// TIA Portal V20 export
TYPE "type_emRelations_em5_cmStatus"
// stored: Access Published, Namespace Unit1
   STRUCT
      cmPnp1stCathodeDetect { S7_SetPoint := 'True'} : "LBC_typeDigitalSignalControlNode";
      cmPnp2ndCathodeDetect { S7_SetPoint := 'True'} : "LBC_typeDigitalSignalControlNode";
      cmCathodeAlignTableElectrodeDetect { S7_SetPoint := 'True'} : "LBC_typeDigitalSignalControlNode";
      cmCathodeNgPnpElectrodeDetect { S7_SetPoint := 'True'} : "LBC_typeDigitalSignalControlNode";
      cmCathodeNgBoxFullSensorDetect { S7_SetPoint := 'True'} : "LBC_typeDigitalSignalControlNode";
      cmCathodeNgBoxDetect { S7_SetPoint := 'True'} : "LBC_typeDigitalSignalControlNode";
      cmCathodeMainPnP1AxisX { ExternalAccessible := 'False'; ExternalVisible := 'False'; ExternalWritable := 'False'} : "LBC_typeAxis64PosControlNode";
      cmCathodeMainPnP2AxisX { ExternalAccessible := 'False'; ExternalVisible := 'False'; ExternalWritable := 'False'} : "LBC_typeAxis64PosControlNode";
      cmCathodeMainPnP1AxisY { ExternalAccessible := 'False'; ExternalVisible := 'False'; ExternalWritable := 'False'} : "LBC_typeAxis64PosControlNode";
      cmCathodeMainPnP1AxisZ { ExternalAccessible := 'False'; ExternalVisible := 'False'; ExternalWritable := 'False'} : "LBC_typeAxis64PosControlNode";
      cmCathodeMainPnP2AxisZ { ExternalAccessible := 'False'; ExternalVisible := 'False'; ExternalWritable := 'False'} : "LBC_typeAxis64PosControlNode";
      cmCathodeAlignTableAxisX { ExternalAccessible := 'False'; ExternalVisible := 'False'; ExternalWritable := 'False'} : "LBC_typeAxis64PosControlNode";
      cmCathodeAlignTableAxisY1 { ExternalAccessible := 'False'; ExternalVisible := 'False'; ExternalWritable := 'False'} : "LBC_typeAxis64PosControlNode";
      cmCathodeAlignTableAxisY2 { ExternalAccessible := 'False'; ExternalVisible := 'False'; ExternalWritable := 'False'} : "LBC_typeAxis64PosControlNode";
      cmCathodeMainPnP1RotaryCwCcw { ExternalAccessible := 'False'; ExternalVisible := 'False'; ExternalWritable := 'False'} : "LBC_typeTwoWayActuatorControlNode";
      cmCathodeMainPnP1SuctionPlateVacuum { ExternalAccessible := 'False'; ExternalVisible := 'False'; ExternalWritable := 'False'} : "LBC_typeTwoWayActuatorControlNode";
      cmCathodeMainPnP2SuctionPlateVacuum { ExternalAccessible := 'False'; ExternalVisible := 'False'; ExternalWritable := 'False'} : "LBC_typeTwoWayActuatorControlNode";
      cmCathodeAlignTableSuctionPlateVacuum { ExternalAccessible := 'False'; ExternalVisible := 'False'; ExternalWritable := 'False'} : "LBC_typeTwoWayActuatorControlNode";
      cmCathodeGlassCleaning { ExternalAccessible := 'False'; ExternalVisible := 'False'; ExternalWritable := 'False'} : "LBC_typeTwoWayActuatorControlNode";
      cmCathodeNgPnpUpDown { ExternalAccessible := 'False'; ExternalVisible := 'False'; ExternalWritable := 'False'} : "LBC_typeTwoWayActuatorControlNode";
      cmCathodeNgPnp1stFwdBwd { ExternalAccessible := 'False'; ExternalVisible := 'False'; ExternalWritable := 'False'} : "LBC_typeTwoWayActuatorControlNode";
      cmCathodeNgPnp2ndFwdBwd { ExternalAccessible := 'False'; ExternalVisible := 'False'; ExternalWritable := 'False'; S7_SetPoint := 'True'} : "LBC_typeTwoWayActuatorControlNode";
      cmCathodeMaintenanceMovingFixFwdBwd { ExternalAccessible := 'False'; ExternalVisible := 'False'; ExternalWritable := 'False'} : "LBC_typeTwoWayActuatorControlNode";
      cmCathodeNgBoxLiftUpDown { ExternalAccessible := 'False'; ExternalVisible := 'False'; ExternalWritable := 'False'; S7_SetPoint := 'True'} : "LBC_typeTwoWayActuatorControlNode";
      cmCathodeNgBoxLockUpDown { ExternalAccessible := 'False'; ExternalVisible := 'False'; ExternalWritable := 'False'; S7_SetPoint := 'True'} : "LBC_typeTwoWayActuatorControlNode";
      cmCathodeNgPnpVaccum { ExternalAccessible := 'False'; ExternalVisible := 'False'; ExternalWritable := 'False'} : "LBC_typeTwoWayActuatorControlNode";
      cmCathodeConveyorCoverFwdBwd { S7_SetPoint := 'True'} : "LBC_typeTwoWayActuatorControlNode";
      cmCathodeConveyorPickUpBlower { S7_SetPoint := 'True'} : "LBC_typeTwoWayActuatorControlNode";
      cmCathodeVisionControllerInterface { ExternalAccessible := 'False'; ExternalVisible := 'False'; ExternalWritable := 'False'} : "LER_typeVisionControlNode";
   END_STRUCT;
   // cmPnp1stCathodeDetect.commands.reset := FALSE;
   // cmPnp1stCathodeDetect.commands.simulation := FALSE;
   // cmPnp1stCathodeDetect.commands.quality := TRUE;
   // cmPnp1stCathodeDetect.monitoring.valid := TRUE;
   // cmPnp1stCathodeDetect.monitoring.busy := TRUE;
   // cmPnp1stCathodeDetect.monitoring.error := FALSE;
   // cmPnp1stCathodeDetect.monitoring.status := 16#0000;
   // cmPnp1stCathodeDetect.monitoring.risingEdge := FALSE;
   // cmPnp1stCathodeDetect.monitoring.fallingEdge := FALSE;
   // cmPnp1stCathodeDetect.monitoring.processValue := FALSE;
   // cmPnp2ndCathodeDetect.commands.reset := FALSE;
   // cmPnp2ndCathodeDetect.commands.simulation := FALSE;
   // cmPnp2ndCathodeDetect.commands.quality := TRUE;
   // cmPnp2ndCathodeDetect.monitoring.valid := TRUE;
   // cmPnp2ndCathodeDetect.monitoring.busy := TRUE;
   // cmPnp2ndCathodeDetect.monitoring.error := FALSE;
   // cmPnp2ndCathodeDetect.monitoring.status := 16#0000;
   // cmPnp2ndCathodeDetect.monitoring.risingEdge := FALSE;
   // cmPnp2ndCathodeDetect.monitoring.fallingEdge := FALSE;
   // cmPnp2ndCathodeDetect.monitoring.processValue := FALSE;
   // cmCathodeAlignTableElectrodeDetect.commands.reset := FALSE;
   // cmCathodeAlignTableElectrodeDetect.commands.simulation := FALSE;
   // cmCathodeAlignTableElectrodeDetect.commands.quality := TRUE;
   // cmCathodeAlignTableElectrodeDetect.monitoring.valid := TRUE;
   // cmCathodeAlignTableElectrodeDetect.monitoring.busy := TRUE;
   // cmCathodeAlignTableElectrodeDetect.monitoring.error := FALSE;
   // cmCathodeAlignTableElectrodeDetect.monitoring.status := 16#0000;
   // cmCathodeAlignTableElectrodeDetect.monitoring.risingEdge := FALSE;
   // cmCathodeAlignTableElectrodeDetect.monitoring.fallingEdge := FALSE;
   // cmCathodeAlignTableElectrodeDetect.monitoring.processValue := FALSE;
   // cmCathodeNgPnpElectrodeDetect.commands.reset := FALSE;
   // cmCathodeNgPnpElectrodeDetect.commands.simulation := FALSE;
   // cmCathodeNgPnpElectrodeDetect.commands.quality := TRUE;
   // cmCathodeNgPnpElectrodeDetect.monitoring.valid := FALSE;
   // cmCathodeNgPnpElectrodeDetect.monitoring.busy := FALSE;
   // cmCathodeNgPnpElectrodeDetect.monitoring.error := FALSE;
   // cmCathodeNgPnpElectrodeDetect.monitoring.status := 16#0000;
   // cmCathodeNgPnpElectrodeDetect.monitoring.risingEdge := FALSE;
   // cmCathodeNgPnpElectrodeDetect.monitoring.fallingEdge := FALSE;
   // cmCathodeNgPnpElectrodeDetect.monitoring.processValue := FALSE;
   // cmCathodeNgBoxFullSensorDetect.commands.reset := FALSE;
   // cmCathodeNgBoxFullSensorDetect.commands.simulation := FALSE;
   // cmCathodeNgBoxFullSensorDetect.commands.quality := TRUE;
   // cmCathodeNgBoxFullSensorDetect.monitoring.valid := TRUE;
   // cmCathodeNgBoxFullSensorDetect.monitoring.busy := TRUE;
   // cmCathodeNgBoxFullSensorDetect.monitoring.error := FALSE;
   // cmCathodeNgBoxFullSensorDetect.monitoring.status := 16#0000;
   // cmCathodeNgBoxFullSensorDetect.monitoring.risingEdge := FALSE;
   // cmCathodeNgBoxFullSensorDetect.monitoring.fallingEdge := FALSE;
   // cmCathodeNgBoxFullSensorDetect.monitoring.processValue := FALSE;
   // cmCathodeNgBoxDetect.commands.reset := FALSE;
   // cmCathodeNgBoxDetect.commands.simulation := FALSE;
   // cmCathodeNgBoxDetect.commands.quality := TRUE;
   // cmCathodeNgBoxDetect.monitoring.valid := TRUE;
   // cmCathodeNgBoxDetect.monitoring.busy := TRUE;
   // cmCathodeNgBoxDetect.monitoring.error := FALSE;
   // cmCathodeNgBoxDetect.monitoring.status := 16#0000;
   // cmCathodeNgBoxDetect.monitoring.risingEdge := FALSE;
   // cmCathodeNgBoxDetect.monitoring.fallingEdge := FALSE;
   // cmCathodeNgBoxDetect.monitoring.processValue := TRUE;
   // cmCathodeMainPnP1AxisX.commandConfiguration.generalSettings.stopOnError := TRUE;
   // cmCathodeMainPnP1AxisX.commandConfiguration.generalSettings.resetWithRestart := FALSE;
   // cmCathodeMainPnP1AxisX.commandConfiguration.generalSettings.abortWaitingSyncCmd := TRUE;
   // cmCathodeMainPnP1AxisX.commandConfiguration.power.startMode := 1;
   // cmCathodeMainPnP1AxisX.commandConfiguration.power.stopMode := 0;
   // cmCathodeMainPnP1AxisX.commandConfiguration.power.syncMotionSimulation := FALSE;
   // cmCathodeMainPnP1AxisX.commandConfiguration.power.syncMotionSimulationExtendedMode := -1;
   // cmCathodeMainPnP1AxisX.commandConfiguration.jog.velocity := 0.0;
   // cmCathodeMainPnP1AxisX.commandConfiguration.jog.acceleration := -1.0;
   // cmCathodeMainPnP1AxisX.commandConfiguration.jog.deceleration := -1.0;
   // cmCathodeMainPnP1AxisX.commandConfiguration.jog.jerk := -1.0;
   // cmCathodeMainPnP1AxisX.commandConfiguration.jog.positionControlled := TRUE;
   // cmCathodeMainPnP1AxisX.commandConfiguration.jog.increment := 0.0;
   // cmCathodeMainPnP1AxisX.commandConfiguration.jog.mode := 0;
   // cmCathodeMainPnP1AxisX.commandConfiguration.moveVelocity.velocity := 0.0;
   // cmCathodeMainPnP1AxisX.commandConfiguration.moveVelocity.acceleration := -1.0;
   // cmCathodeMainPnP1AxisX.commandConfiguration.moveVelocity.deceleration := -1.0;
   // cmCathodeMainPnP1AxisX.commandConfiguration.moveVelocity.jerk := -1.0;
   // cmCathodeMainPnP1AxisX.commandConfiguration.moveVelocity.direction := 0;
   // cmCathodeMainPnP1AxisX.commandConfiguration.moveVelocity.positionControlled := TRUE;
   // cmCathodeMainPnP1AxisX.commandConfiguration.moveVelocity.velocityChangeOnTheFly := FALSE;
   // cmCathodeMainPnP1AxisX.commandConfiguration.stop.deceleration := -1.0;
   // cmCathodeMainPnP1AxisX.commandConfiguration.stop.jerk := -1.0;
   // cmCathodeMainPnP1AxisX.commandConfiguration.stop.abortAcceleration := FALSE;
   // cmCathodeMainPnP1AxisX.commandConfiguration.fastStop.deceleration := -1.0;
   // cmCathodeMainPnP1AxisX.commandConfiguration.fastStop.jerk := -1.0;
   // cmCathodeMainPnP1AxisX.commandConfiguration.fastStop.abortAcceleration := FALSE;
   // cmCathodeMainPnP1AxisX.commandConfiguration.fastStop.replaceStopPossible := FALSE;
   // cmCathodeMainPnP1AxisX.commandConfiguration.torqueLimiting.limit := -1.0;
   // cmCathodeMainPnP1AxisX.commandConfiguration.torqueLimiting.mode := 0;
   // cmCathodeMainPnP1AxisX.commandConfiguration.homing.position := 0.0;
   // cmCathodeMainPnP1AxisX.commandConfiguration.homing.mode := 0;
   // cmCathodeMainPnP1AxisX.commandConfiguration.homing.sensor := 0;
   // cmCathodeMainPnP1AxisX.commandConfiguration.homing.extendedMode := -1;
   // cmCathodeMainPnP1AxisX.commandConfiguration.homing.extendedModeTorqueLimit := 0.0;
   // cmCathodeMainPnP1AxisX.commandConfiguration.homing.extendedModeTargetPosition := 0.0;
   // cmCathodeMainPnP1AxisX.commandConfiguration.posRelative.distance := 0.0;
   // cmCathodeMainPnP1AxisX.commandConfiguration.posRelative.velocity := -1.0;
   // cmCathodeMainPnP1AxisX.commandConfiguration.posRelative.acceleration := -1.0;
   // cmCathodeMainPnP1AxisX.commandConfiguration.posRelative.deceleration := -1.0;
   // cmCathodeMainPnP1AxisX.commandConfiguration.posRelative.jerk := -1.0;
   // cmCathodeMainPnP1AxisX.commandConfiguration.posRelative.direction := 0;
   // cmCathodeMainPnP1AxisX.commandConfiguration.posAbsolute.position := 0.0;
   // cmCathodeMainPnP1AxisX.commandConfiguration.posAbsolute.velocity := -1.0;
   // cmCathodeMainPnP1AxisX.commandConfiguration.posAbsolute.acceleration := -1.0;
   // cmCathodeMainPnP1AxisX.commandConfiguration.posAbsolute.deceleration := -1.0;
   // cmCathodeMainPnP1AxisX.commandConfiguration.posAbsolute.jerk := -1.0;
   // cmCathodeMainPnP1AxisX.commandConfiguration.posAbsolute.direction := 1;
   // cmCathodeMainPnP1AxisX.commandConfiguration.posAbsolute.positionChangeOnTheFly := FALSE;
   // cmCathodeMainPnP1AxisX.commandConfiguration.posAbsolute.velocityChangeOnTheFly := FALSE;
   // cmCathodeMainPnP1AxisX.commandConfiguration.posSuperimposed.distance := 0.0;
   // cmCathodeMainPnP1AxisX.commandConfiguration.posSuperimposed.velocityDiff := -1.0;
   // cmCathodeMainPnP1AxisX.commandConfiguration.posSuperimposed.acceleration := -1.0;
   // cmCathodeMainPnP1AxisX.commandConfiguration.posSuperimposed.deceleration := -1.0;
   // cmCathodeMainPnP1AxisX.commandConfiguration.posSuperimposed.jerk := -1.0;
   // cmCathodeMainPnP1AxisX.commandConfiguration.posSuperimposed.direction := 0;
   // cmCathodeMainPnP1AxisX.commandConfiguration.haltSuperimposed.deceleration := -1.0;
   // cmCathodeMainPnP1AxisX.commandConfiguration.haltSuperimposed.jerk := -1.0;
   // cmCathodeMainPnP1AxisX.commandConfiguration.haltSuperimposed.abortAcceleration := FALSE;
   // cmCathodeMainPnP1AxisX.commandConfiguration.gearInRelative.ratioNumerator := 1;
   // cmCathodeMainPnP1AxisX.commandConfiguration.gearInRelative.ratioDenominator := 1;
   // cmCathodeMainPnP1AxisX.commandConfiguration.gearInRelative.acceleration := -1.0;
   // cmCathodeMainPnP1AxisX.commandConfiguration.gearInRelative.deceleration := -1.0;
   // cmCathodeMainPnP1AxisX.commandConfiguration.gearInRelative.jerk := -1.0;
   // cmCathodeMainPnP1AxisX.commandConfiguration.gearInRelative.ratioChangeOnTheFly := FALSE;
   // cmCathodeMainPnP1AxisX.commandConfiguration.gearInAbsolute.ratioNumerator := 1;
   // cmCathodeMainPnP1AxisX.commandConfiguration.gearInAbsolute.ratioDenominator := 1;
   // cmCathodeMainPnP1AxisX.commandConfiguration.gearInAbsolute.masterSyncPosition := 0.0;
   // cmCathodeMainPnP1AxisX.commandConfiguration.gearInAbsolute.slaveSyncPosition := 0.0;
   // cmCathodeMainPnP1AxisX.commandConfiguration.gearInAbsolute.syncProfileReference := 1;
   // cmCathodeMainPnP1AxisX.commandConfiguration.gearInAbsolute.masterStartDistance := 0.0;
   // cmCathodeMainPnP1AxisX.commandConfiguration.gearInAbsolute.velocity := -1.0;
   // cmCathodeMainPnP1AxisX.commandConfiguration.gearInAbsolute.acceleration := -1.0;
   // cmCathodeMainPnP1AxisX.commandConfiguration.gearInAbsolute.deceleration := -1.0;
   // cmCathodeMainPnP1AxisX.commandConfiguration.gearInAbsolute.jerk := -1.0;
   // cmCathodeMainPnP1AxisX.commandConfiguration.gearInAbsolute.syncDirection := 1;
   // cmCathodeMainPnP1AxisX.commandConfiguration.gearInAbsolute.ratioChangeOnTheFly := FALSE;
   // cmCathodeMainPnP1AxisX.commandConfiguration.gearInVelocity.continuousUpdate := FALSE;
   // cmCathodeMainPnP1AxisX.commandConfiguration.gearInVelocity.ratioNumerator := 1;
   // cmCathodeMainPnP1AxisX.commandConfiguration.gearInVelocity.ratioDenominator := 1;
   // cmCathodeMainPnP1AxisX.commandConfiguration.gearInVelocity.acceleration := -1.0;
   // cmCathodeMainPnP1AxisX.commandConfiguration.gearInVelocity.deceleration := -1.0;
   // cmCathodeMainPnP1AxisX.commandConfiguration.gearInVelocity.jerk := -1.0;
   // cmCathodeMainPnP1AxisX.commandConfiguration.gearInVelocity.positionControlled := FALSE;
   // cmCathodeMainPnP1AxisX.commandConfiguration.camIn.masterOffset := 0.0;
   // cmCathodeMainPnP1AxisX.commandConfiguration.camIn.slaveOffset := 0.0;
   // cmCathodeMainPnP1AxisX.commandConfiguration.camIn.masterScaling := 1.0;
   // cmCathodeMainPnP1AxisX.commandConfiguration.camIn.slaveScaling := 1.0;
   // cmCathodeMainPnP1AxisX.commandConfiguration.camIn.masterSyncPosition := 0.0;
   // cmCathodeMainPnP1AxisX.commandConfiguration.camIn.syncProfileReference := 1;
   // cmCathodeMainPnP1AxisX.commandConfiguration.camIn.masterStartDistance := 0.0;
   // cmCathodeMainPnP1AxisX.commandConfiguration.camIn.velocity := -1.0;
   // cmCathodeMainPnP1AxisX.commandConfiguration.camIn.acceleration := -1.0;
   // cmCathodeMainPnP1AxisX.commandConfiguration.camIn.deceleration := -1.0;
   // cmCathodeMainPnP1AxisX.commandConfiguration.camIn.jerk := -1.0;
   // cmCathodeMainPnP1AxisX.commandConfiguration.camIn.applicationMode := 0;
   // cmCathodeMainPnP1AxisX.commandConfiguration.camIn.syncDirection := 1;
   // cmCathodeMainPnP1AxisX.commandConfiguration.gearOutCamOut.slavePosition := 0.0;
   // cmCathodeMainPnP1AxisX.commandConfiguration.gearOutCamOut.syncProfileReference := 1;
   // cmCathodeMainPnP1AxisX.commandConfiguration.gearOutCamOut.masterStopDistance := 0.0;
   // cmCathodeMainPnP1AxisX.commandConfiguration.gearOutCamOut.deceleration := -1.0;
   // cmCathodeMainPnP1AxisX.commandConfiguration.gearOutCamOut.jerk := -1.0;
   // cmCathodeMainPnP1AxisX.commandConfiguration.gearOutCamOut.syncOutDirection := 3;
   // cmCathodeMainPnP1AxisX.commandConfiguration.gearOutCamOut.gearOutCamOutMode := -1;
   // cmCathodeMainPnP1AxisX.commandConfiguration.phasing.phaseShift := 0.0;
   // cmCathodeMainPnP1AxisX.commandConfiguration.phasing.velocity := -1.0;
   // cmCathodeMainPnP1AxisX.commandConfiguration.phasing.acceleration := -1.0;
   // cmCathodeMainPnP1AxisX.commandConfiguration.phasing.deceleration := -1.0;
   // cmCathodeMainPnP1AxisX.commandConfiguration.phasing.jerk := -1.0;
   // cmCathodeMainPnP1AxisX.commandConfiguration.phasing.profileReference := 0;
   // cmCathodeMainPnP1AxisX.commandConfiguration.phasing.phasingDistance := 0.0;
   // cmCathodeMainPnP1AxisX.commandConfiguration.phasing.startPosition := 0.0;
   // cmCathodeMainPnP1AxisX.commandConfiguration.phasing.direction := 3;
   // cmCathodeMainPnP1AxisX.commandConfiguration.phasing.phaseAbsolute := TRUE;
   // cmCathodeMainPnP1AxisX.commandConfiguration.phasing.phaseShiftChangeOnTheFly := FALSE;
   // cmCathodeMainPnP1AxisX.commandConfiguration.offset.offset := 0.0;
   // cmCathodeMainPnP1AxisX.commandConfiguration.offset.profileReference := 1;
   // cmCathodeMainPnP1AxisX.commandConfiguration.offset.offsetDistance := 0.0;
   // cmCathodeMainPnP1AxisX.commandConfiguration.offset.startPosition := 0.0;
   // cmCathodeMainPnP1AxisX.commandConfiguration.offset.direction := 3;
   // cmCathodeMainPnP1AxisX.commandConfiguration.offset.offsetAbsolute := TRUE;
   // cmCathodeMainPnP1AxisX.commandConfiguration.offset.offsetChangeOnTheFly := FALSE;
   // cmCathodeMainPnP1AxisX.commands.enableAxis := FALSE;
   // cmCathodeMainPnP1AxisX.commands.resetAxis := FALSE;
   // cmCathodeMainPnP1AxisX.commands.openBrake := FALSE;
   // cmCathodeMainPnP1AxisX.commands.jogForward := FALSE;
   // cmCathodeMainPnP1AxisX.commands.jogBackward := FALSE;
   // cmCathodeMainPnP1AxisX.commands.moveVelocity := FALSE;
   // cmCathodeMainPnP1AxisX.commands.stop := FALSE;
   // cmCathodeMainPnP1AxisX.commands.fastStop := FALSE;
   // cmCathodeMainPnP1AxisX.commands.torqueLimiting := FALSE;
   // cmCathodeMainPnP1AxisX.commands.homing := FALSE;
   // cmCathodeMainPnP1AxisX.commands.posRelative := FALSE;
   // cmCathodeMainPnP1AxisX.commands.posAbsolute := FALSE;
   // cmCathodeMainPnP1AxisX.commands.posSuperimposed := FALSE;
   // cmCathodeMainPnP1AxisX.commands.haltSuperimposed := FALSE;
   // cmCathodeMainPnP1AxisX.commands.selectSetPosition := -1;
   // cmCathodeMainPnP1AxisX.commands.reset := FALSE;
   // cmCathodeMainPnP1AxisX.monitoring.valid := FALSE;
   // cmCathodeMainPnP1AxisX.monitoring.busy := TRUE;
   // cmCathodeMainPnP1AxisX.monitoring.error := TRUE;
   // cmCathodeMainPnP1AxisX.monitoring.status := 16#8600;
   // cmCathodeMainPnP1AxisX.monitoring.subfunctionStatus := 16#8001;
   // cmCathodeMainPnP1AxisX.monitoring.axisEnabled := FALSE;
   // cmCathodeMainPnP1AxisX.monitoring.resetActive := FALSE;
   // cmCathodeMainPnP1AxisX.monitoring.inVelocity := FALSE;
   // cmCathodeMainPnP1AxisX.monitoring.inLimitation := FALSE;
   // cmCathodeMainPnP1AxisX.monitoring.inClamping := FALSE;
   // cmCathodeMainPnP1AxisX.monitoring.startSync := FALSE;
   // cmCathodeMainPnP1AxisX.monitoring.inSync := FALSE;
   // cmCathodeMainPnP1AxisX.monitoring.inSimulation := FALSE;
   // cmCathodeMainPnP1AxisX.monitoring.jogSelected := FALSE;
   // cmCathodeMainPnP1AxisX.monitoring.moveVelocitySelected := FALSE;
   // cmCathodeMainPnP1AxisX.monitoring.stopSelected := FALSE;
   // cmCathodeMainPnP1AxisX.monitoring.fastStopSelected := FALSE;
   // cmCathodeMainPnP1AxisX.monitoring.torqueLimitingSelected := FALSE;
   // cmCathodeMainPnP1AxisX.monitoring.homingSelected := FALSE;
   // cmCathodeMainPnP1AxisX.monitoring.posRelativeSelected := FALSE;
   // cmCathodeMainPnP1AxisX.monitoring.posAbsoluteSelected := FALSE;
   // cmCathodeMainPnP1AxisX.monitoring.posSuperimposedSelected := FALSE;
   // cmCathodeMainPnP1AxisX.monitoring.haltSuperimposedSelected := FALSE;
   // cmCathodeMainPnP1AxisX.monitoring.commandBusy := FALSE;
   // cmCathodeMainPnP1AxisX.monitoring.commandDone := FALSE;
   // cmCathodeMainPnP1AxisX.monitoring.commandAborted := FALSE;
   // cmCathodeMainPnP1AxisX.monitoring.homingCommandBusy := FALSE;
   // cmCathodeMainPnP1AxisX.monitoring.homingCommandDone := FALSE;
   // cmCathodeMainPnP1AxisX.monitoring.homingCommandAborted := FALSE;
   // cmCathodeMainPnP1AxisX.monitoring.superimposedBusy := FALSE;
   // cmCathodeMainPnP1AxisX.monitoring.superimposedDone := FALSE;
   // cmCathodeMainPnP1AxisX.monitoring.superimposedAborted := FALSE;
   // cmCathodeMainPnP1AxisX.monitoring.actualPosition := 0.048;
   // cmCathodeMainPnP1AxisX.monitoring.actualSpeed := 0.0;
   // cmCathodeMainPnP1AxisX.monitoring.speedUnit := 1062;
   // cmCathodeMainPnP1AxisX.monitoring.positionUnit := 1013;
   // cmCathodeMainPnP1AxisX.monitoring.axisType := 1;
   // cmCathodeMainPnP1AxisX.monitoring.interlockGeneralOut := TRUE;
   // cmCathodeMainPnP1AxisX.monitoring.interlockJogForwardOut := TRUE;
   // cmCathodeMainPnP1AxisX.monitoring.interlockJogBackwardOut := TRUE;
   // cmCathodeMainPnP2AxisX.commandConfiguration.generalSettings.stopOnError := TRUE;
   // cmCathodeMainPnP2AxisX.commandConfiguration.generalSettings.resetWithRestart := FALSE;
   // cmCathodeMainPnP2AxisX.commandConfiguration.generalSettings.abortWaitingSyncCmd := TRUE;
   // cmCathodeMainPnP2AxisX.commandConfiguration.power.startMode := 1;
   // cmCathodeMainPnP2AxisX.commandConfiguration.power.stopMode := 0;
   // cmCathodeMainPnP2AxisX.commandConfiguration.power.syncMotionSimulation := FALSE;
   // cmCathodeMainPnP2AxisX.commandConfiguration.power.syncMotionSimulationExtendedMode := -1;
   // cmCathodeMainPnP2AxisX.commandConfiguration.jog.velocity := 0.0;
   // cmCathodeMainPnP2AxisX.commandConfiguration.jog.acceleration := -1.0;
   // cmCathodeMainPnP2AxisX.commandConfiguration.jog.deceleration := -1.0;
   // cmCathodeMainPnP2AxisX.commandConfiguration.jog.jerk := -1.0;
   // cmCathodeMainPnP2AxisX.commandConfiguration.jog.positionControlled := TRUE;
   // cmCathodeMainPnP2AxisX.commandConfiguration.jog.increment := 0.0;
   // cmCathodeMainPnP2AxisX.commandConfiguration.jog.mode := 0;
   // cmCathodeMainPnP2AxisX.commandConfiguration.moveVelocity.velocity := 0.0;
   // cmCathodeMainPnP2AxisX.commandConfiguration.moveVelocity.acceleration := -1.0;
   // cmCathodeMainPnP2AxisX.commandConfiguration.moveVelocity.deceleration := -1.0;
   // cmCathodeMainPnP2AxisX.commandConfiguration.moveVelocity.jerk := -1.0;
   // cmCathodeMainPnP2AxisX.commandConfiguration.moveVelocity.direction := 0;
   // cmCathodeMainPnP2AxisX.commandConfiguration.moveVelocity.positionControlled := TRUE;
   // cmCathodeMainPnP2AxisX.commandConfiguration.moveVelocity.velocityChangeOnTheFly := FALSE;
   // cmCathodeMainPnP2AxisX.commandConfiguration.stop.deceleration := -1.0;
   // cmCathodeMainPnP2AxisX.commandConfiguration.stop.jerk := -1.0;
   // cmCathodeMainPnP2AxisX.commandConfiguration.stop.abortAcceleration := FALSE;
   // cmCathodeMainPnP2AxisX.commandConfiguration.fastStop.deceleration := -1.0;
   // cmCathodeMainPnP2AxisX.commandConfiguration.fastStop.jerk := -1.0;
   // cmCathodeMainPnP2AxisX.commandConfiguration.fastStop.abortAcceleration := FALSE;
   // cmCathodeMainPnP2AxisX.commandConfiguration.fastStop.replaceStopPossible := FALSE;
   // cmCathodeMainPnP2AxisX.commandConfiguration.torqueLimiting.limit := -1.0;
   // cmCathodeMainPnP2AxisX.commandConfiguration.torqueLimiting.mode := 0;
   // cmCathodeMainPnP2AxisX.commandConfiguration.homing.position := 0.0;
   // cmCathodeMainPnP2AxisX.commandConfiguration.homing.mode := 0;
   // cmCathodeMainPnP2AxisX.commandConfiguration.homing.sensor := 0;
   // cmCathodeMainPnP2AxisX.commandConfiguration.homing.extendedMode := -1;
   // cmCathodeMainPnP2AxisX.commandConfiguration.homing.extendedModeTorqueLimit := 0.0;
   // cmCathodeMainPnP2AxisX.commandConfiguration.homing.extendedModeTargetPosition := 0.0;
   // cmCathodeMainPnP2AxisX.commandConfiguration.posRelative.distance := 0.0;
   // cmCathodeMainPnP2AxisX.commandConfiguration.posRelative.velocity := -1.0;
   // cmCathodeMainPnP2AxisX.commandConfiguration.posRelative.acceleration := -1.0;
   // cmCathodeMainPnP2AxisX.commandConfiguration.posRelative.deceleration := -1.0;
   // cmCathodeMainPnP2AxisX.commandConfiguration.posRelative.jerk := -1.0;
   // cmCathodeMainPnP2AxisX.commandConfiguration.posRelative.direction := 0;
   // cmCathodeMainPnP2AxisX.commandConfiguration.posAbsolute.position := 0.0;
   // cmCathodeMainPnP2AxisX.commandConfiguration.posAbsolute.velocity := -1.0;
   // cmCathodeMainPnP2AxisX.commandConfiguration.posAbsolute.acceleration := -1.0;
   // cmCathodeMainPnP2AxisX.commandConfiguration.posAbsolute.deceleration := -1.0;
   // cmCathodeMainPnP2AxisX.commandConfiguration.posAbsolute.jerk := -1.0;
   // cmCathodeMainPnP2AxisX.commandConfiguration.posAbsolute.direction := 1;
   // cmCathodeMainPnP2AxisX.commandConfiguration.posAbsolute.positionChangeOnTheFly := FALSE;
   // cmCathodeMainPnP2AxisX.commandConfiguration.posAbsolute.velocityChangeOnTheFly := FALSE;
   // cmCathodeMainPnP2AxisX.commandConfiguration.posSuperimposed.distance := 0.0;
   // cmCathodeMainPnP2AxisX.commandConfiguration.posSuperimposed.velocityDiff := -1.0;
   // cmCathodeMainPnP2AxisX.commandConfiguration.posSuperimposed.acceleration := -1.0;
   // cmCathodeMainPnP2AxisX.commandConfiguration.posSuperimposed.deceleration := -1.0;
   // cmCathodeMainPnP2AxisX.commandConfiguration.posSuperimposed.jerk := -1.0;
   // cmCathodeMainPnP2AxisX.commandConfiguration.posSuperimposed.direction := 0;
   // cmCathodeMainPnP2AxisX.commandConfiguration.haltSuperimposed.deceleration := -1.0;
   // cmCathodeMainPnP2AxisX.commandConfiguration.haltSuperimposed.jerk := -1.0;
   // cmCathodeMainPnP2AxisX.commandConfiguration.haltSuperimposed.abortAcceleration := FALSE;
   // cmCathodeMainPnP2AxisX.commandConfiguration.gearInRelative.ratioNumerator := 1;
   // cmCathodeMainPnP2AxisX.commandConfiguration.gearInRelative.ratioDenominator := 1;
   // cmCathodeMainPnP2AxisX.commandConfiguration.gearInRelative.acceleration := -1.0;
   // cmCathodeMainPnP2AxisX.commandConfiguration.gearInRelative.deceleration := -1.0;
   // cmCathodeMainPnP2AxisX.commandConfiguration.gearInRelative.jerk := -1.0;
   // cmCathodeMainPnP2AxisX.commandConfiguration.gearInRelative.ratioChangeOnTheFly := FALSE;
   // cmCathodeMainPnP2AxisX.commandConfiguration.gearInAbsolute.ratioNumerator := 1;
   // cmCathodeMainPnP2AxisX.commandConfiguration.gearInAbsolute.ratioDenominator := 1;
   // cmCathodeMainPnP2AxisX.commandConfiguration.gearInAbsolute.masterSyncPosition := 0.0;
   // cmCathodeMainPnP2AxisX.commandConfiguration.gearInAbsolute.slaveSyncPosition := 0.0;
   // cmCathodeMainPnP2AxisX.commandConfiguration.gearInAbsolute.syncProfileReference := 1;
   // cmCathodeMainPnP2AxisX.commandConfiguration.gearInAbsolute.masterStartDistance := 0.0;
   // cmCathodeMainPnP2AxisX.commandConfiguration.gearInAbsolute.velocity := -1.0;
   // cmCathodeMainPnP2AxisX.commandConfiguration.gearInAbsolute.acceleration := -1.0;
   // cmCathodeMainPnP2AxisX.commandConfiguration.gearInAbsolute.deceleration := -1.0;
   // cmCathodeMainPnP2AxisX.commandConfiguration.gearInAbsolute.jerk := -1.0;
   // cmCathodeMainPnP2AxisX.commandConfiguration.gearInAbsolute.syncDirection := 1;
   // cmCathodeMainPnP2AxisX.commandConfiguration.gearInAbsolute.ratioChangeOnTheFly := FALSE;
   // cmCathodeMainPnP2AxisX.commandConfiguration.gearInVelocity.continuousUpdate := FALSE;
   // cmCathodeMainPnP2AxisX.commandConfiguration.gearInVelocity.ratioNumerator := 1;
   // cmCathodeMainPnP2AxisX.commandConfiguration.gearInVelocity.ratioDenominator := 1;
   // cmCathodeMainPnP2AxisX.commandConfiguration.gearInVelocity.acceleration := -1.0;
   // cmCathodeMainPnP2AxisX.commandConfiguration.gearInVelocity.deceleration := -1.0;
   // cmCathodeMainPnP2AxisX.commandConfiguration.gearInVelocity.jerk := -1.0;
   // cmCathodeMainPnP2AxisX.commandConfiguration.gearInVelocity.positionControlled := FALSE;
   // cmCathodeMainPnP2AxisX.commandConfiguration.camIn.masterOffset := 0.0;
   // cmCathodeMainPnP2AxisX.commandConfiguration.camIn.slaveOffset := 0.0;
   // cmCathodeMainPnP2AxisX.commandConfiguration.camIn.masterScaling := 1.0;
   // cmCathodeMainPnP2AxisX.commandConfiguration.camIn.slaveScaling := 1.0;
   // cmCathodeMainPnP2AxisX.commandConfiguration.camIn.masterSyncPosition := 0.0;
   // cmCathodeMainPnP2AxisX.commandConfiguration.camIn.syncProfileReference := 1;
   // cmCathodeMainPnP2AxisX.commandConfiguration.camIn.masterStartDistance := 0.0;
   // cmCathodeMainPnP2AxisX.commandConfiguration.camIn.velocity := -1.0;
   // cmCathodeMainPnP2AxisX.commandConfiguration.camIn.acceleration := -1.0;
   // cmCathodeMainPnP2AxisX.commandConfiguration.camIn.deceleration := -1.0;
   // cmCathodeMainPnP2AxisX.commandConfiguration.camIn.jerk := -1.0;
   // cmCathodeMainPnP2AxisX.commandConfiguration.camIn.applicationMode := 0;
   // cmCathodeMainPnP2AxisX.commandConfiguration.camIn.syncDirection := 1;
   // cmCathodeMainPnP2AxisX.commandConfiguration.gearOutCamOut.slavePosition := 0.0;
   // cmCathodeMainPnP2AxisX.commandConfiguration.gearOutCamOut.syncProfileReference := 1;
   // cmCathodeMainPnP2AxisX.commandConfiguration.gearOutCamOut.masterStopDistance := 0.0;
   // cmCathodeMainPnP2AxisX.commandConfiguration.gearOutCamOut.deceleration := -1.0;
   // cmCathodeMainPnP2AxisX.commandConfiguration.gearOutCamOut.jerk := -1.0;
   // cmCathodeMainPnP2AxisX.commandConfiguration.gearOutCamOut.syncOutDirection := 3;
   // cmCathodeMainPnP2AxisX.commandConfiguration.gearOutCamOut.gearOutCamOutMode := -1;
   // cmCathodeMainPnP2AxisX.commandConfiguration.phasing.phaseShift := 0.0;
   // cmCathodeMainPnP2AxisX.commandConfiguration.phasing.velocity := -1.0;
   // cmCathodeMainPnP2AxisX.commandConfiguration.phasing.acceleration := -1.0;
   // cmCathodeMainPnP2AxisX.commandConfiguration.phasing.deceleration := -1.0;
   // cmCathodeMainPnP2AxisX.commandConfiguration.phasing.jerk := -1.0;
   // cmCathodeMainPnP2AxisX.commandConfiguration.phasing.profileReference := 0;
   // cmCathodeMainPnP2AxisX.commandConfiguration.phasing.phasingDistance := 0.0;
   // cmCathodeMainPnP2AxisX.commandConfiguration.phasing.startPosition := 0.0;
   // cmCathodeMainPnP2AxisX.commandConfiguration.phasing.direction := 3;
   // cmCathodeMainPnP2AxisX.commandConfiguration.phasing.phaseAbsolute := TRUE;
   // cmCathodeMainPnP2AxisX.commandConfiguration.phasing.phaseShiftChangeOnTheFly := FALSE;
   // cmCathodeMainPnP2AxisX.commandConfiguration.offset.offset := 0.0;
   // cmCathodeMainPnP2AxisX.commandConfiguration.offset.profileReference := 1;
   // cmCathodeMainPnP2AxisX.commandConfiguration.offset.offsetDistance := 0.0;
   // cmCathodeMainPnP2AxisX.commandConfiguration.offset.startPosition := 0.0;
   // cmCathodeMainPnP2AxisX.commandConfiguration.offset.direction := 3;
   // cmCathodeMainPnP2AxisX.commandConfiguration.offset.offsetAbsolute := TRUE;
   // cmCathodeMainPnP2AxisX.commandConfiguration.offset.offsetChangeOnTheFly := FALSE;
   // cmCathodeMainPnP2AxisX.commands.enableAxis := FALSE;
   // cmCathodeMainPnP2AxisX.commands.resetAxis := FALSE;
   // cmCathodeMainPnP2AxisX.commands.openBrake := FALSE;
   // cmCathodeMainPnP2AxisX.commands.jogForward := FALSE;
   // cmCathodeMainPnP2AxisX.commands.jogBackward := FALSE;
   // cmCathodeMainPnP2AxisX.commands.moveVelocity := FALSE;
   // cmCathodeMainPnP2AxisX.commands.stop := FALSE;
   // cmCathodeMainPnP2AxisX.commands.fastStop := FALSE;
   // cmCathodeMainPnP2AxisX.commands.torqueLimiting := FALSE;
   // cmCathodeMainPnP2AxisX.commands.homing := FALSE;
   // cmCathodeMainPnP2AxisX.commands.posRelative := FALSE;
   // cmCathodeMainPnP2AxisX.commands.posAbsolute := FALSE;
   // cmCathodeMainPnP2AxisX.commands.posSuperimposed := FALSE;
   // cmCathodeMainPnP2AxisX.commands.haltSuperimposed := FALSE;
   // cmCathodeMainPnP2AxisX.commands.selectSetPosition := -1;
   // cmCathodeMainPnP2AxisX.commands.reset := FALSE;
   // cmCathodeMainPnP2AxisX.monitoring.valid := FALSE;
   // cmCathodeMainPnP2AxisX.monitoring.busy := TRUE;
   // cmCathodeMainPnP2AxisX.monitoring.error := TRUE;
   // cmCathodeMainPnP2AxisX.monitoring.status := 16#8600;
   // cmCathodeMainPnP2AxisX.monitoring.subfunctionStatus := 16#8001;
   // cmCathodeMainPnP2AxisX.monitoring.axisEnabled := FALSE;
   // cmCathodeMainPnP2AxisX.monitoring.resetActive := FALSE;
   // cmCathodeMainPnP2AxisX.monitoring.inVelocity := FALSE;
   // cmCathodeMainPnP2AxisX.monitoring.inLimitation := FALSE;
   // cmCathodeMainPnP2AxisX.monitoring.inClamping := FALSE;
   // cmCathodeMainPnP2AxisX.monitoring.startSync := FALSE;
   // cmCathodeMainPnP2AxisX.monitoring.inSync := FALSE;
   // cmCathodeMainPnP2AxisX.monitoring.inSimulation := FALSE;
   // cmCathodeMainPnP2AxisX.monitoring.jogSelected := FALSE;
   // cmCathodeMainPnP2AxisX.monitoring.moveVelocitySelected := FALSE;
   // cmCathodeMainPnP2AxisX.monitoring.stopSelected := FALSE;
   // cmCathodeMainPnP2AxisX.monitoring.fastStopSelected := FALSE;
   // cmCathodeMainPnP2AxisX.monitoring.torqueLimitingSelected := FALSE;
   // cmCathodeMainPnP2AxisX.monitoring.homingSelected := FALSE;
   // cmCathodeMainPnP2AxisX.monitoring.posRelativeSelected := FALSE;
   // cmCathodeMainPnP2AxisX.monitoring.posAbsoluteSelected := FALSE;
   // cmCathodeMainPnP2AxisX.monitoring.posSuperimposedSelected := FALSE;
   // cmCathodeMainPnP2AxisX.monitoring.haltSuperimposedSelected := FALSE;
   // cmCathodeMainPnP2AxisX.monitoring.commandBusy := FALSE;
   // cmCathodeMainPnP2AxisX.monitoring.commandDone := FALSE;
   // cmCathodeMainPnP2AxisX.monitoring.commandAborted := FALSE;
   // cmCathodeMainPnP2AxisX.monitoring.homingCommandBusy := FALSE;
   // cmCathodeMainPnP2AxisX.monitoring.homingCommandDone := FALSE;
   // cmCathodeMainPnP2AxisX.monitoring.homingCommandAborted := FALSE;
   // cmCathodeMainPnP2AxisX.monitoring.superimposedBusy := FALSE;
   // cmCathodeMainPnP2AxisX.monitoring.superimposedDone := FALSE;
   // cmCathodeMainPnP2AxisX.monitoring.superimposedAborted := FALSE;
   // cmCathodeMainPnP2AxisX.monitoring.actualPosition := -11.988;
   // cmCathodeMainPnP2AxisX.monitoring.actualSpeed := -0.000333333333333333;
   // cmCathodeMainPnP2AxisX.monitoring.speedUnit := 1062;
   // cmCathodeMainPnP2AxisX.monitoring.positionUnit := 1013;
   // cmCathodeMainPnP2AxisX.monitoring.axisType := 1;
   // cmCathodeMainPnP2AxisX.monitoring.interlockGeneralOut := TRUE;
   // cmCathodeMainPnP2AxisX.monitoring.interlockJogForwardOut := TRUE;
   // cmCathodeMainPnP2AxisX.monitoring.interlockJogBackwardOut := TRUE;
   // cmCathodeMainPnP1AxisY.commandConfiguration.generalSettings.stopOnError := TRUE;
   // cmCathodeMainPnP1AxisY.commandConfiguration.generalSettings.resetWithRestart := FALSE;
   // cmCathodeMainPnP1AxisY.commandConfiguration.generalSettings.abortWaitingSyncCmd := TRUE;
   // cmCathodeMainPnP1AxisY.commandConfiguration.power.startMode := 1;
   // cmCathodeMainPnP1AxisY.commandConfiguration.power.stopMode := 0;
   // cmCathodeMainPnP1AxisY.commandConfiguration.power.syncMotionSimulation := FALSE;
   // cmCathodeMainPnP1AxisY.commandConfiguration.power.syncMotionSimulationExtendedMode := -1;
   // cmCathodeMainPnP1AxisY.commandConfiguration.jog.velocity := 0.0;
   // cmCathodeMainPnP1AxisY.commandConfiguration.jog.acceleration := -1.0;
   // cmCathodeMainPnP1AxisY.commandConfiguration.jog.deceleration := -1.0;
   // cmCathodeMainPnP1AxisY.commandConfiguration.jog.jerk := -1.0;
   // cmCathodeMainPnP1AxisY.commandConfiguration.jog.positionControlled := TRUE;
   // cmCathodeMainPnP1AxisY.commandConfiguration.jog.increment := 0.0;
   // cmCathodeMainPnP1AxisY.commandConfiguration.jog.mode := 0;
   // cmCathodeMainPnP1AxisY.commandConfiguration.moveVelocity.velocity := 0.0;
   // cmCathodeMainPnP1AxisY.commandConfiguration.moveVelocity.acceleration := -1.0;
   // cmCathodeMainPnP1AxisY.commandConfiguration.moveVelocity.deceleration := -1.0;
   // cmCathodeMainPnP1AxisY.commandConfiguration.moveVelocity.jerk := -1.0;
   // cmCathodeMainPnP1AxisY.commandConfiguration.moveVelocity.direction := 0;
   // cmCathodeMainPnP1AxisY.commandConfiguration.moveVelocity.positionControlled := TRUE;
   // cmCathodeMainPnP1AxisY.commandConfiguration.moveVelocity.velocityChangeOnTheFly := FALSE;
   // cmCathodeMainPnP1AxisY.commandConfiguration.stop.deceleration := -1.0;
   // cmCathodeMainPnP1AxisY.commandConfiguration.stop.jerk := -1.0;
   // cmCathodeMainPnP1AxisY.commandConfiguration.stop.abortAcceleration := FALSE;
   // cmCathodeMainPnP1AxisY.commandConfiguration.fastStop.deceleration := -1.0;
   // cmCathodeMainPnP1AxisY.commandConfiguration.fastStop.jerk := -1.0;
   // cmCathodeMainPnP1AxisY.commandConfiguration.fastStop.abortAcceleration := FALSE;
   // cmCathodeMainPnP1AxisY.commandConfiguration.fastStop.replaceStopPossible := FALSE;
   // cmCathodeMainPnP1AxisY.commandConfiguration.torqueLimiting.limit := -1.0;
   // cmCathodeMainPnP1AxisY.commandConfiguration.torqueLimiting.mode := 0;
   // cmCathodeMainPnP1AxisY.commandConfiguration.homing.position := 0.0;
   // cmCathodeMainPnP1AxisY.commandConfiguration.homing.mode := 0;
   // cmCathodeMainPnP1AxisY.commandConfiguration.homing.sensor := 0;
   // cmCathodeMainPnP1AxisY.commandConfiguration.homing.extendedMode := -1;
   // cmCathodeMainPnP1AxisY.commandConfiguration.homing.extendedModeTorqueLimit := 0.0;
   // cmCathodeMainPnP1AxisY.commandConfiguration.homing.extendedModeTargetPosition := 0.0;
   // cmCathodeMainPnP1AxisY.commandConfiguration.posRelative.distance := 0.0;
   // cmCathodeMainPnP1AxisY.commandConfiguration.posRelative.velocity := -1.0;
   // cmCathodeMainPnP1AxisY.commandConfiguration.posRelative.acceleration := -1.0;
   // cmCathodeMainPnP1AxisY.commandConfiguration.posRelative.deceleration := -1.0;
   // cmCathodeMainPnP1AxisY.commandConfiguration.posRelative.jerk := -1.0;
   // cmCathodeMainPnP1AxisY.commandConfiguration.posRelative.direction := 0;
   // cmCathodeMainPnP1AxisY.commandConfiguration.posAbsolute.position := 0.0;
   // cmCathodeMainPnP1AxisY.commandConfiguration.posAbsolute.velocity := -1.0;
   // cmCathodeMainPnP1AxisY.commandConfiguration.posAbsolute.acceleration := -1.0;
   // cmCathodeMainPnP1AxisY.commandConfiguration.posAbsolute.deceleration := -1.0;
   // cmCathodeMainPnP1AxisY.commandConfiguration.posAbsolute.jerk := -1.0;
   // cmCathodeMainPnP1AxisY.commandConfiguration.posAbsolute.direction := 1;
   // cmCathodeMainPnP1AxisY.commandConfiguration.posAbsolute.positionChangeOnTheFly := FALSE;
   // cmCathodeMainPnP1AxisY.commandConfiguration.posAbsolute.velocityChangeOnTheFly := FALSE;
   // cmCathodeMainPnP1AxisY.commandConfiguration.posSuperimposed.distance := 0.0;
   // cmCathodeMainPnP1AxisY.commandConfiguration.posSuperimposed.velocityDiff := -1.0;
   // cmCathodeMainPnP1AxisY.commandConfiguration.posSuperimposed.acceleration := -1.0;
   // cmCathodeMainPnP1AxisY.commandConfiguration.posSuperimposed.deceleration := -1.0;
   // cmCathodeMainPnP1AxisY.commandConfiguration.posSuperimposed.jerk := -1.0;
   // cmCathodeMainPnP1AxisY.commandConfiguration.posSuperimposed.direction := 0;
   // cmCathodeMainPnP1AxisY.commandConfiguration.haltSuperimposed.deceleration := -1.0;
   // cmCathodeMainPnP1AxisY.commandConfiguration.haltSuperimposed.jerk := -1.0;
   // cmCathodeMainPnP1AxisY.commandConfiguration.haltSuperimposed.abortAcceleration := FALSE;
   // cmCathodeMainPnP1AxisY.commandConfiguration.gearInRelative.ratioNumerator := 1;
   // cmCathodeMainPnP1AxisY.commandConfiguration.gearInRelative.ratioDenominator := 1;
   // cmCathodeMainPnP1AxisY.commandConfiguration.gearInRelative.acceleration := -1.0;
   // cmCathodeMainPnP1AxisY.commandConfiguration.gearInRelative.deceleration := -1.0;
   // cmCathodeMainPnP1AxisY.commandConfiguration.gearInRelative.jerk := -1.0;
   // cmCathodeMainPnP1AxisY.commandConfiguration.gearInRelative.ratioChangeOnTheFly := FALSE;
   // cmCathodeMainPnP1AxisY.commandConfiguration.gearInAbsolute.ratioNumerator := 1;
   // cmCathodeMainPnP1AxisY.commandConfiguration.gearInAbsolute.ratioDenominator := 1;
   // cmCathodeMainPnP1AxisY.commandConfiguration.gearInAbsolute.masterSyncPosition := 0.0;
   // cmCathodeMainPnP1AxisY.commandConfiguration.gearInAbsolute.slaveSyncPosition := 0.0;
   // cmCathodeMainPnP1AxisY.commandConfiguration.gearInAbsolute.syncProfileReference := 1;
   // cmCathodeMainPnP1AxisY.commandConfiguration.gearInAbsolute.masterStartDistance := 0.0;
   // cmCathodeMainPnP1AxisY.commandConfiguration.gearInAbsolute.velocity := -1.0;
   // cmCathodeMainPnP1AxisY.commandConfiguration.gearInAbsolute.acceleration := -1.0;
   // cmCathodeMainPnP1AxisY.commandConfiguration.gearInAbsolute.deceleration := -1.0;
   // cmCathodeMainPnP1AxisY.commandConfiguration.gearInAbsolute.jerk := -1.0;
   // cmCathodeMainPnP1AxisY.commandConfiguration.gearInAbsolute.syncDirection := 1;
   // cmCathodeMainPnP1AxisY.commandConfiguration.gearInAbsolute.ratioChangeOnTheFly := FALSE;
   // cmCathodeMainPnP1AxisY.commandConfiguration.gearInVelocity.continuousUpdate := FALSE;
   // cmCathodeMainPnP1AxisY.commandConfiguration.gearInVelocity.ratioNumerator := 1;
   // cmCathodeMainPnP1AxisY.commandConfiguration.gearInVelocity.ratioDenominator := 1;
   // cmCathodeMainPnP1AxisY.commandConfiguration.gearInVelocity.acceleration := -1.0;
   // cmCathodeMainPnP1AxisY.commandConfiguration.gearInVelocity.deceleration := -1.0;
   // cmCathodeMainPnP1AxisY.commandConfiguration.gearInVelocity.jerk := -1.0;
   // cmCathodeMainPnP1AxisY.commandConfiguration.gearInVelocity.positionControlled := FALSE;
   // cmCathodeMainPnP1AxisY.commandConfiguration.camIn.masterOffset := 0.0;
   // cmCathodeMainPnP1AxisY.commandConfiguration.camIn.slaveOffset := 0.0;
   // cmCathodeMainPnP1AxisY.commandConfiguration.camIn.masterScaling := 1.0;
   // cmCathodeMainPnP1AxisY.commandConfiguration.camIn.slaveScaling := 1.0;
   // cmCathodeMainPnP1AxisY.commandConfiguration.camIn.masterSyncPosition := 0.0;
   // cmCathodeMainPnP1AxisY.commandConfiguration.camIn.syncProfileReference := 1;
   // cmCathodeMainPnP1AxisY.commandConfiguration.camIn.masterStartDistance := 0.0;
   // cmCathodeMainPnP1AxisY.commandConfiguration.camIn.velocity := -1.0;
   // cmCathodeMainPnP1AxisY.commandConfiguration.camIn.acceleration := -1.0;
   // cmCathodeMainPnP1AxisY.commandConfiguration.camIn.deceleration := -1.0;
   // cmCathodeMainPnP1AxisY.commandConfiguration.camIn.jerk := -1.0;
   // cmCathodeMainPnP1AxisY.commandConfiguration.camIn.applicationMode := 0;
   // cmCathodeMainPnP1AxisY.commandConfiguration.camIn.syncDirection := 1;
   // cmCathodeMainPnP1AxisY.commandConfiguration.gearOutCamOut.slavePosition := 0.0;
   // cmCathodeMainPnP1AxisY.commandConfiguration.gearOutCamOut.syncProfileReference := 1;
   // cmCathodeMainPnP1AxisY.commandConfiguration.gearOutCamOut.masterStopDistance := 0.0;
   // cmCathodeMainPnP1AxisY.commandConfiguration.gearOutCamOut.deceleration := -1.0;
   // cmCathodeMainPnP1AxisY.commandConfiguration.gearOutCamOut.jerk := -1.0;
   // cmCathodeMainPnP1AxisY.commandConfiguration.gearOutCamOut.syncOutDirection := 3;
   // cmCathodeMainPnP1AxisY.commandConfiguration.gearOutCamOut.gearOutCamOutMode := -1;
   // cmCathodeMainPnP1AxisY.commandConfiguration.phasing.phaseShift := 0.0;
   // cmCathodeMainPnP1AxisY.commandConfiguration.phasing.velocity := -1.0;
   // cmCathodeMainPnP1AxisY.commandConfiguration.phasing.acceleration := -1.0;
   // cmCathodeMainPnP1AxisY.commandConfiguration.phasing.deceleration := -1.0;
   // cmCathodeMainPnP1AxisY.commandConfiguration.phasing.jerk := -1.0;
   // cmCathodeMainPnP1AxisY.commandConfiguration.phasing.profileReference := 0;
   // cmCathodeMainPnP1AxisY.commandConfiguration.phasing.phasingDistance := 0.0;
   // cmCathodeMainPnP1AxisY.commandConfiguration.phasing.startPosition := 0.0;
   // cmCathodeMainPnP1AxisY.commandConfiguration.phasing.direction := 3;
   // cmCathodeMainPnP1AxisY.commandConfiguration.phasing.phaseAbsolute := TRUE;
   // cmCathodeMainPnP1AxisY.commandConfiguration.phasing.phaseShiftChangeOnTheFly := FALSE;
   // cmCathodeMainPnP1AxisY.commandConfiguration.offset.offset := 0.0;
   // cmCathodeMainPnP1AxisY.commandConfiguration.offset.profileReference := 1;
   // cmCathodeMainPnP1AxisY.commandConfiguration.offset.offsetDistance := 0.0;
   // cmCathodeMainPnP1AxisY.commandConfiguration.offset.startPosition := 0.0;
   // cmCathodeMainPnP1AxisY.commandConfiguration.offset.direction := 3;
   // cmCathodeMainPnP1AxisY.commandConfiguration.offset.offsetAbsolute := TRUE;
   // cmCathodeMainPnP1AxisY.commandConfiguration.offset.offsetChangeOnTheFly := FALSE;
   // cmCathodeMainPnP1AxisY.commands.enableAxis := FALSE;
   // cmCathodeMainPnP1AxisY.commands.resetAxis := FALSE;
   // cmCathodeMainPnP1AxisY.commands.openBrake := FALSE;
   // cmCathodeMainPnP1AxisY.commands.jogForward := FALSE;
   // cmCathodeMainPnP1AxisY.commands.jogBackward := FALSE;
   // cmCathodeMainPnP1AxisY.commands.moveVelocity := FALSE;
   // cmCathodeMainPnP1AxisY.commands.stop := FALSE;
   // cmCathodeMainPnP1AxisY.commands.fastStop := FALSE;
   // cmCathodeMainPnP1AxisY.commands.torqueLimiting := FALSE;
   // cmCathodeMainPnP1AxisY.commands.homing := FALSE;
   // cmCathodeMainPnP1AxisY.commands.posRelative := FALSE;
   // cmCathodeMainPnP1AxisY.commands.posAbsolute := FALSE;
   // cmCathodeMainPnP1AxisY.commands.posSuperimposed := FALSE;
   // cmCathodeMainPnP1AxisY.commands.haltSuperimposed := FALSE;
   // cmCathodeMainPnP1AxisY.commands.selectSetPosition := -1;
   // cmCathodeMainPnP1AxisY.commands.reset := FALSE;
   // cmCathodeMainPnP1AxisY.monitoring.valid := FALSE;
   // cmCathodeMainPnP1AxisY.monitoring.busy := TRUE;
   // cmCathodeMainPnP1AxisY.monitoring.error := TRUE;
   // cmCathodeMainPnP1AxisY.monitoring.status := 16#8600;
   // cmCathodeMainPnP1AxisY.monitoring.subfunctionStatus := 16#8001;
   // cmCathodeMainPnP1AxisY.monitoring.axisEnabled := FALSE;
   // cmCathodeMainPnP1AxisY.monitoring.resetActive := FALSE;
   // cmCathodeMainPnP1AxisY.monitoring.inVelocity := FALSE;
   // cmCathodeMainPnP1AxisY.monitoring.inLimitation := FALSE;
   // cmCathodeMainPnP1AxisY.monitoring.inClamping := FALSE;
   // cmCathodeMainPnP1AxisY.monitoring.startSync := FALSE;
   // cmCathodeMainPnP1AxisY.monitoring.inSync := FALSE;
   // cmCathodeMainPnP1AxisY.monitoring.inSimulation := FALSE;
   // cmCathodeMainPnP1AxisY.monitoring.jogSelected := FALSE;
   // cmCathodeMainPnP1AxisY.monitoring.moveVelocitySelected := FALSE;
   // cmCathodeMainPnP1AxisY.monitoring.stopSelected := FALSE;
   // cmCathodeMainPnP1AxisY.monitoring.fastStopSelected := FALSE;
   // cmCathodeMainPnP1AxisY.monitoring.torqueLimitingSelected := FALSE;
   // cmCathodeMainPnP1AxisY.monitoring.homingSelected := FALSE;
   // cmCathodeMainPnP1AxisY.monitoring.posRelativeSelected := FALSE;
   // cmCathodeMainPnP1AxisY.monitoring.posAbsoluteSelected := FALSE;
   // cmCathodeMainPnP1AxisY.monitoring.posSuperimposedSelected := FALSE;
   // cmCathodeMainPnP1AxisY.monitoring.haltSuperimposedSelected := FALSE;
   // cmCathodeMainPnP1AxisY.monitoring.commandBusy := FALSE;
   // cmCathodeMainPnP1AxisY.monitoring.commandDone := FALSE;
   // cmCathodeMainPnP1AxisY.monitoring.commandAborted := FALSE;
   // cmCathodeMainPnP1AxisY.monitoring.homingCommandBusy := FALSE;
   // cmCathodeMainPnP1AxisY.monitoring.homingCommandDone := FALSE;
   // cmCathodeMainPnP1AxisY.monitoring.homingCommandAborted := FALSE;
   // cmCathodeMainPnP1AxisY.monitoring.superimposedBusy := FALSE;
   // cmCathodeMainPnP1AxisY.monitoring.superimposedDone := FALSE;
   // cmCathodeMainPnP1AxisY.monitoring.superimposedAborted := FALSE;
   // cmCathodeMainPnP1AxisY.monitoring.actualPosition := 0.0;
   // cmCathodeMainPnP1AxisY.monitoring.actualSpeed := 0.0;
   // cmCathodeMainPnP1AxisY.monitoring.speedUnit := 1062;
   // cmCathodeMainPnP1AxisY.monitoring.positionUnit := 1013;
   // cmCathodeMainPnP1AxisY.monitoring.axisType := 1;
   // cmCathodeMainPnP1AxisY.monitoring.interlockGeneralOut := TRUE;
   // cmCathodeMainPnP1AxisY.monitoring.interlockJogForwardOut := TRUE;
   // cmCathodeMainPnP1AxisY.monitoring.interlockJogBackwardOut := TRUE;
   // cmCathodeMainPnP1AxisZ.commandConfiguration.generalSettings.stopOnError := TRUE;
   // cmCathodeMainPnP1AxisZ.commandConfiguration.generalSettings.resetWithRestart := FALSE;
   // cmCathodeMainPnP1AxisZ.commandConfiguration.generalSettings.abortWaitingSyncCmd := TRUE;
   // cmCathodeMainPnP1AxisZ.commandConfiguration.power.startMode := 1;
   // cmCathodeMainPnP1AxisZ.commandConfiguration.power.stopMode := 0;
   // cmCathodeMainPnP1AxisZ.commandConfiguration.power.syncMotionSimulation := FALSE;
   // cmCathodeMainPnP1AxisZ.commandConfiguration.power.syncMotionSimulationExtendedMode := -1;
   // cmCathodeMainPnP1AxisZ.commandConfiguration.jog.velocity := 10.0;
   // cmCathodeMainPnP1AxisZ.commandConfiguration.jog.acceleration := -1.0;
   // cmCathodeMainPnP1AxisZ.commandConfiguration.jog.deceleration := -1.0;
   // cmCathodeMainPnP1AxisZ.commandConfiguration.jog.jerk := -1.0;
   // cmCathodeMainPnP1AxisZ.commandConfiguration.jog.positionControlled := TRUE;
   // cmCathodeMainPnP1AxisZ.commandConfiguration.jog.increment := 0.0;
   // cmCathodeMainPnP1AxisZ.commandConfiguration.jog.mode := 0;
   // cmCathodeMainPnP1AxisZ.commandConfiguration.moveVelocity.velocity := 0.0;
   // cmCathodeMainPnP1AxisZ.commandConfiguration.moveVelocity.acceleration := -1.0;
   // cmCathodeMainPnP1AxisZ.commandConfiguration.moveVelocity.deceleration := -1.0;
   // cmCathodeMainPnP1AxisZ.commandConfiguration.moveVelocity.jerk := -1.0;
   // cmCathodeMainPnP1AxisZ.commandConfiguration.moveVelocity.direction := 0;
   // cmCathodeMainPnP1AxisZ.commandConfiguration.moveVelocity.positionControlled := TRUE;
   // cmCathodeMainPnP1AxisZ.commandConfiguration.moveVelocity.velocityChangeOnTheFly := FALSE;
   // cmCathodeMainPnP1AxisZ.commandConfiguration.stop.deceleration := -1.0;
   // cmCathodeMainPnP1AxisZ.commandConfiguration.stop.jerk := -1.0;
   // cmCathodeMainPnP1AxisZ.commandConfiguration.stop.abortAcceleration := FALSE;
   // cmCathodeMainPnP1AxisZ.commandConfiguration.fastStop.deceleration := -1.0;
   // cmCathodeMainPnP1AxisZ.commandConfiguration.fastStop.jerk := -1.0;
   // cmCathodeMainPnP1AxisZ.commandConfiguration.fastStop.abortAcceleration := FALSE;
   // cmCathodeMainPnP1AxisZ.commandConfiguration.fastStop.replaceStopPossible := FALSE;
   // cmCathodeMainPnP1AxisZ.commandConfiguration.torqueLimiting.limit := -1.0;
   // cmCathodeMainPnP1AxisZ.commandConfiguration.torqueLimiting.mode := 0;
   // cmCathodeMainPnP1AxisZ.commandConfiguration.homing.position := 0.0;
   // cmCathodeMainPnP1AxisZ.commandConfiguration.homing.mode := 0;
   // cmCathodeMainPnP1AxisZ.commandConfiguration.homing.sensor := 0;
   // cmCathodeMainPnP1AxisZ.commandConfiguration.homing.extendedMode := -1;
   // cmCathodeMainPnP1AxisZ.commandConfiguration.homing.extendedModeTorqueLimit := 0.0;
   // cmCathodeMainPnP1AxisZ.commandConfiguration.homing.extendedModeTargetPosition := 0.0;
   // cmCathodeMainPnP1AxisZ.commandConfiguration.posRelative.distance := 0.0;
   // cmCathodeMainPnP1AxisZ.commandConfiguration.posRelative.velocity := -1.0;
   // cmCathodeMainPnP1AxisZ.commandConfiguration.posRelative.acceleration := -1.0;
   // cmCathodeMainPnP1AxisZ.commandConfiguration.posRelative.deceleration := -1.0;
   // cmCathodeMainPnP1AxisZ.commandConfiguration.posRelative.jerk := -1.0;
   // cmCathodeMainPnP1AxisZ.commandConfiguration.posRelative.direction := 0;
   // cmCathodeMainPnP1AxisZ.commandConfiguration.posAbsolute.position := 0.0;
   // cmCathodeMainPnP1AxisZ.commandConfiguration.posAbsolute.velocity := -1.0;
   // cmCathodeMainPnP1AxisZ.commandConfiguration.posAbsolute.acceleration := -1.0;
   // cmCathodeMainPnP1AxisZ.commandConfiguration.posAbsolute.deceleration := -1.0;
   // cmCathodeMainPnP1AxisZ.commandConfiguration.posAbsolute.jerk := -1.0;
   // cmCathodeMainPnP1AxisZ.commandConfiguration.posAbsolute.direction := 1;
   // cmCathodeMainPnP1AxisZ.commandConfiguration.posAbsolute.positionChangeOnTheFly := FALSE;
   // cmCathodeMainPnP1AxisZ.commandConfiguration.posAbsolute.velocityChangeOnTheFly := FALSE;
   // cmCathodeMainPnP1AxisZ.commandConfiguration.posSuperimposed.distance := 0.0;
   // cmCathodeMainPnP1AxisZ.commandConfiguration.posSuperimposed.velocityDiff := -1.0;
   // cmCathodeMainPnP1AxisZ.commandConfiguration.posSuperimposed.acceleration := -1.0;
   // cmCathodeMainPnP1AxisZ.commandConfiguration.posSuperimposed.deceleration := -1.0;
   // cmCathodeMainPnP1AxisZ.commandConfiguration.posSuperimposed.jerk := -1.0;
   // cmCathodeMainPnP1AxisZ.commandConfiguration.posSuperimposed.direction := 0;
   // cmCathodeMainPnP1AxisZ.commandConfiguration.haltSuperimposed.deceleration := -1.0;
   // cmCathodeMainPnP1AxisZ.commandConfiguration.haltSuperimposed.jerk := -1.0;
   // cmCathodeMainPnP1AxisZ.commandConfiguration.haltSuperimposed.abortAcceleration := FALSE;
   // cmCathodeMainPnP1AxisZ.commandConfiguration.gearInRelative.ratioNumerator := 1;
   // cmCathodeMainPnP1AxisZ.commandConfiguration.gearInRelative.ratioDenominator := 1;
   // cmCathodeMainPnP1AxisZ.commandConfiguration.gearInRelative.acceleration := -1.0;
   // cmCathodeMainPnP1AxisZ.commandConfiguration.gearInRelative.deceleration := -1.0;
   // cmCathodeMainPnP1AxisZ.commandConfiguration.gearInRelative.jerk := -1.0;
   // cmCathodeMainPnP1AxisZ.commandConfiguration.gearInRelative.ratioChangeOnTheFly := FALSE;
   // cmCathodeMainPnP1AxisZ.commandConfiguration.gearInAbsolute.ratioNumerator := 1;
   // cmCathodeMainPnP1AxisZ.commandConfiguration.gearInAbsolute.ratioDenominator := 1;
   // cmCathodeMainPnP1AxisZ.commandConfiguration.gearInAbsolute.masterSyncPosition := 0.0;
   // cmCathodeMainPnP1AxisZ.commandConfiguration.gearInAbsolute.slaveSyncPosition := 0.0;
   // cmCathodeMainPnP1AxisZ.commandConfiguration.gearInAbsolute.syncProfileReference := 1;
   // cmCathodeMainPnP1AxisZ.commandConfiguration.gearInAbsolute.masterStartDistance := 0.0;
   // cmCathodeMainPnP1AxisZ.commandConfiguration.gearInAbsolute.velocity := -1.0;
   // cmCathodeMainPnP1AxisZ.commandConfiguration.gearInAbsolute.acceleration := -1.0;
   // cmCathodeMainPnP1AxisZ.commandConfiguration.gearInAbsolute.deceleration := -1.0;
   // cmCathodeMainPnP1AxisZ.commandConfiguration.gearInAbsolute.jerk := -1.0;
   // cmCathodeMainPnP1AxisZ.commandConfiguration.gearInAbsolute.syncDirection := 1;
   // cmCathodeMainPnP1AxisZ.commandConfiguration.gearInAbsolute.ratioChangeOnTheFly := FALSE;
   // cmCathodeMainPnP1AxisZ.commandConfiguration.gearInVelocity.continuousUpdate := FALSE;
   // cmCathodeMainPnP1AxisZ.commandConfiguration.gearInVelocity.ratioNumerator := 1;
   // cmCathodeMainPnP1AxisZ.commandConfiguration.gearInVelocity.ratioDenominator := 1;
   // cmCathodeMainPnP1AxisZ.commandConfiguration.gearInVelocity.acceleration := -1.0;
   // cmCathodeMainPnP1AxisZ.commandConfiguration.gearInVelocity.deceleration := -1.0;
   // cmCathodeMainPnP1AxisZ.commandConfiguration.gearInVelocity.jerk := -1.0;
   // cmCathodeMainPnP1AxisZ.commandConfiguration.gearInVelocity.positionControlled := FALSE;
   // cmCathodeMainPnP1AxisZ.commandConfiguration.camIn.masterOffset := 0.0;
   // cmCathodeMainPnP1AxisZ.commandConfiguration.camIn.slaveOffset := 0.0;
   // cmCathodeMainPnP1AxisZ.commandConfiguration.camIn.masterScaling := 1.0;
   // cmCathodeMainPnP1AxisZ.commandConfiguration.camIn.slaveScaling := 1.0;
   // cmCathodeMainPnP1AxisZ.commandConfiguration.camIn.masterSyncPosition := 0.0;
   // cmCathodeMainPnP1AxisZ.commandConfiguration.camIn.syncProfileReference := 1;
   // cmCathodeMainPnP1AxisZ.commandConfiguration.camIn.masterStartDistance := 0.0;
   // cmCathodeMainPnP1AxisZ.commandConfiguration.camIn.velocity := -1.0;
   // cmCathodeMainPnP1AxisZ.commandConfiguration.camIn.acceleration := -1.0;
   // cmCathodeMainPnP1AxisZ.commandConfiguration.camIn.deceleration := -1.0;
   // cmCathodeMainPnP1AxisZ.commandConfiguration.camIn.jerk := -1.0;
   // cmCathodeMainPnP1AxisZ.commandConfiguration.camIn.applicationMode := 0;
   // cmCathodeMainPnP1AxisZ.commandConfiguration.camIn.syncDirection := 1;
   // cmCathodeMainPnP1AxisZ.commandConfiguration.gearOutCamOut.slavePosition := 0.0;
   // cmCathodeMainPnP1AxisZ.commandConfiguration.gearOutCamOut.syncProfileReference := 1;
   // cmCathodeMainPnP1AxisZ.commandConfiguration.gearOutCamOut.masterStopDistance := 0.0;
   // cmCathodeMainPnP1AxisZ.commandConfiguration.gearOutCamOut.deceleration := -1.0;
   // cmCathodeMainPnP1AxisZ.commandConfiguration.gearOutCamOut.jerk := -1.0;
   // cmCathodeMainPnP1AxisZ.commandConfiguration.gearOutCamOut.syncOutDirection := 3;
   // cmCathodeMainPnP1AxisZ.commandConfiguration.gearOutCamOut.gearOutCamOutMode := -1;
   // cmCathodeMainPnP1AxisZ.commandConfiguration.phasing.phaseShift := 0.0;
   // cmCathodeMainPnP1AxisZ.commandConfiguration.phasing.velocity := -1.0;
   // cmCathodeMainPnP1AxisZ.commandConfiguration.phasing.acceleration := -1.0;
   // cmCathodeMainPnP1AxisZ.commandConfiguration.phasing.deceleration := -1.0;
   // cmCathodeMainPnP1AxisZ.commandConfiguration.phasing.jerk := -1.0;
   // cmCathodeMainPnP1AxisZ.commandConfiguration.phasing.profileReference := 0;
   // cmCathodeMainPnP1AxisZ.commandConfiguration.phasing.phasingDistance := 0.0;
   // cmCathodeMainPnP1AxisZ.commandConfiguration.phasing.startPosition := 0.0;
   // cmCathodeMainPnP1AxisZ.commandConfiguration.phasing.direction := 3;
   // cmCathodeMainPnP1AxisZ.commandConfiguration.phasing.phaseAbsolute := TRUE;
   // cmCathodeMainPnP1AxisZ.commandConfiguration.phasing.phaseShiftChangeOnTheFly := FALSE;
   // cmCathodeMainPnP1AxisZ.commandConfiguration.offset.offset := 0.0;
   // cmCathodeMainPnP1AxisZ.commandConfiguration.offset.profileReference := 1;
   // cmCathodeMainPnP1AxisZ.commandConfiguration.offset.offsetDistance := 0.0;
   // cmCathodeMainPnP1AxisZ.commandConfiguration.offset.startPosition := 0.0;
   // cmCathodeMainPnP1AxisZ.commandConfiguration.offset.direction := 3;
   // cmCathodeMainPnP1AxisZ.commandConfiguration.offset.offsetAbsolute := TRUE;
   // cmCathodeMainPnP1AxisZ.commandConfiguration.offset.offsetChangeOnTheFly := FALSE;
   // cmCathodeMainPnP1AxisZ.commands.enableAxis := FALSE;
   // cmCathodeMainPnP1AxisZ.commands.resetAxis := FALSE;
   // cmCathodeMainPnP1AxisZ.commands.openBrake := FALSE;
   // cmCathodeMainPnP1AxisZ.commands.jogForward := FALSE;
   // cmCathodeMainPnP1AxisZ.commands.jogBackward := FALSE;
   // cmCathodeMainPnP1AxisZ.commands.moveVelocity := FALSE;
   // cmCathodeMainPnP1AxisZ.commands.stop := FALSE;
   // cmCathodeMainPnP1AxisZ.commands.fastStop := FALSE;
   // cmCathodeMainPnP1AxisZ.commands.torqueLimiting := FALSE;
   // cmCathodeMainPnP1AxisZ.commands.homing := FALSE;
   // cmCathodeMainPnP1AxisZ.commands.posRelative := FALSE;
   // cmCathodeMainPnP1AxisZ.commands.posAbsolute := FALSE;
   // cmCathodeMainPnP1AxisZ.commands.posSuperimposed := FALSE;
   // cmCathodeMainPnP1AxisZ.commands.haltSuperimposed := FALSE;
   // cmCathodeMainPnP1AxisZ.commands.selectSetPosition := -1;
   // cmCathodeMainPnP1AxisZ.commands.reset := FALSE;
   // cmCathodeMainPnP1AxisZ.monitoring.valid := FALSE;
   // cmCathodeMainPnP1AxisZ.monitoring.busy := TRUE;
   // cmCathodeMainPnP1AxisZ.monitoring.error := TRUE;
   // cmCathodeMainPnP1AxisZ.monitoring.status := 16#8600;
   // cmCathodeMainPnP1AxisZ.monitoring.subfunctionStatus := 16#8001;
   // cmCathodeMainPnP1AxisZ.monitoring.axisEnabled := FALSE;
   // cmCathodeMainPnP1AxisZ.monitoring.resetActive := FALSE;
   // cmCathodeMainPnP1AxisZ.monitoring.inVelocity := FALSE;
   // cmCathodeMainPnP1AxisZ.monitoring.inLimitation := FALSE;
   // cmCathodeMainPnP1AxisZ.monitoring.inClamping := FALSE;
   // cmCathodeMainPnP1AxisZ.monitoring.startSync := FALSE;
   // cmCathodeMainPnP1AxisZ.monitoring.inSync := FALSE;
   // cmCathodeMainPnP1AxisZ.monitoring.inSimulation := FALSE;
   // cmCathodeMainPnP1AxisZ.monitoring.jogSelected := FALSE;
   // cmCathodeMainPnP1AxisZ.monitoring.moveVelocitySelected := FALSE;
   // cmCathodeMainPnP1AxisZ.monitoring.stopSelected := FALSE;
   // cmCathodeMainPnP1AxisZ.monitoring.fastStopSelected := FALSE;
   // cmCathodeMainPnP1AxisZ.monitoring.torqueLimitingSelected := FALSE;
   // cmCathodeMainPnP1AxisZ.monitoring.homingSelected := FALSE;
   // cmCathodeMainPnP1AxisZ.monitoring.posRelativeSelected := FALSE;
   // cmCathodeMainPnP1AxisZ.monitoring.posAbsoluteSelected := FALSE;
   // cmCathodeMainPnP1AxisZ.monitoring.posSuperimposedSelected := FALSE;
   // cmCathodeMainPnP1AxisZ.monitoring.haltSuperimposedSelected := FALSE;
   // cmCathodeMainPnP1AxisZ.monitoring.commandBusy := FALSE;
   // cmCathodeMainPnP1AxisZ.monitoring.commandDone := FALSE;
   // cmCathodeMainPnP1AxisZ.monitoring.commandAborted := FALSE;
   // cmCathodeMainPnP1AxisZ.monitoring.homingCommandBusy := FALSE;
   // cmCathodeMainPnP1AxisZ.monitoring.homingCommandDone := FALSE;
   // cmCathodeMainPnP1AxisZ.monitoring.homingCommandAborted := FALSE;
   // cmCathodeMainPnP1AxisZ.monitoring.superimposedBusy := FALSE;
   // cmCathodeMainPnP1AxisZ.monitoring.superimposedDone := FALSE;
   // cmCathodeMainPnP1AxisZ.monitoring.superimposedAborted := FALSE;
   // cmCathodeMainPnP1AxisZ.monitoring.actualPosition := 5.609;
   // cmCathodeMainPnP1AxisZ.monitoring.actualSpeed := 0.0;
   // cmCathodeMainPnP1AxisZ.monitoring.speedUnit := 1062;
   // cmCathodeMainPnP1AxisZ.monitoring.positionUnit := 1013;
   // cmCathodeMainPnP1AxisZ.monitoring.axisType := 1;
   // cmCathodeMainPnP1AxisZ.monitoring.interlockGeneralOut := TRUE;
   // cmCathodeMainPnP1AxisZ.monitoring.interlockJogForwardOut := TRUE;
   // cmCathodeMainPnP1AxisZ.monitoring.interlockJogBackwardOut := TRUE;
   // cmCathodeMainPnP2AxisZ.commandConfiguration.generalSettings.stopOnError := TRUE;
   // cmCathodeMainPnP2AxisZ.commandConfiguration.generalSettings.resetWithRestart := FALSE;
   // cmCathodeMainPnP2AxisZ.commandConfiguration.generalSettings.abortWaitingSyncCmd := TRUE;
   // cmCathodeMainPnP2AxisZ.commandConfiguration.power.startMode := 1;
   // cmCathodeMainPnP2AxisZ.commandConfiguration.power.stopMode := 0;
   // cmCathodeMainPnP2AxisZ.commandConfiguration.power.syncMotionSimulation := FALSE;
   // cmCathodeMainPnP2AxisZ.commandConfiguration.power.syncMotionSimulationExtendedMode := -1;
   // cmCathodeMainPnP2AxisZ.commandConfiguration.jog.velocity := 10.0;
   // cmCathodeMainPnP2AxisZ.commandConfiguration.jog.acceleration := -1.0;
   // cmCathodeMainPnP2AxisZ.commandConfiguration.jog.deceleration := -1.0;
   // cmCathodeMainPnP2AxisZ.commandConfiguration.jog.jerk := -1.0;
   // cmCathodeMainPnP2AxisZ.commandConfiguration.jog.positionControlled := TRUE;
   // cmCathodeMainPnP2AxisZ.commandConfiguration.jog.increment := 0.0;
   // cmCathodeMainPnP2AxisZ.commandConfiguration.jog.mode := 0;
   // cmCathodeMainPnP2AxisZ.commandConfiguration.moveVelocity.velocity := 0.0;
   // cmCathodeMainPnP2AxisZ.commandConfiguration.moveVelocity.acceleration := -1.0;
   // cmCathodeMainPnP2AxisZ.commandConfiguration.moveVelocity.deceleration := -1.0;
   // cmCathodeMainPnP2AxisZ.commandConfiguration.moveVelocity.jerk := -1.0;
   // cmCathodeMainPnP2AxisZ.commandConfiguration.moveVelocity.direction := 0;
   // cmCathodeMainPnP2AxisZ.commandConfiguration.moveVelocity.positionControlled := TRUE;
   // cmCathodeMainPnP2AxisZ.commandConfiguration.moveVelocity.velocityChangeOnTheFly := FALSE;
   // cmCathodeMainPnP2AxisZ.commandConfiguration.stop.deceleration := -1.0;
   // cmCathodeMainPnP2AxisZ.commandConfiguration.stop.jerk := -1.0;
   // cmCathodeMainPnP2AxisZ.commandConfiguration.stop.abortAcceleration := FALSE;
   // cmCathodeMainPnP2AxisZ.commandConfiguration.fastStop.deceleration := -1.0;
   // cmCathodeMainPnP2AxisZ.commandConfiguration.fastStop.jerk := -1.0;
   // cmCathodeMainPnP2AxisZ.commandConfiguration.fastStop.abortAcceleration := FALSE;
   // cmCathodeMainPnP2AxisZ.commandConfiguration.fastStop.replaceStopPossible := FALSE;
   // cmCathodeMainPnP2AxisZ.commandConfiguration.torqueLimiting.limit := -1.0;
   // cmCathodeMainPnP2AxisZ.commandConfiguration.torqueLimiting.mode := 0;
   // cmCathodeMainPnP2AxisZ.commandConfiguration.homing.position := 0.0;
   // cmCathodeMainPnP2AxisZ.commandConfiguration.homing.mode := 0;
   // cmCathodeMainPnP2AxisZ.commandConfiguration.homing.sensor := 0;
   // cmCathodeMainPnP2AxisZ.commandConfiguration.homing.extendedMode := -1;
   // cmCathodeMainPnP2AxisZ.commandConfiguration.homing.extendedModeTorqueLimit := 0.0;
   // cmCathodeMainPnP2AxisZ.commandConfiguration.homing.extendedModeTargetPosition := 0.0;
   // cmCathodeMainPnP2AxisZ.commandConfiguration.posRelative.distance := 0.0;
   // cmCathodeMainPnP2AxisZ.commandConfiguration.posRelative.velocity := -1.0;
   // cmCathodeMainPnP2AxisZ.commandConfiguration.posRelative.acceleration := -1.0;
   // cmCathodeMainPnP2AxisZ.commandConfiguration.posRelative.deceleration := -1.0;
   // cmCathodeMainPnP2AxisZ.commandConfiguration.posRelative.jerk := -1.0;
   // cmCathodeMainPnP2AxisZ.commandConfiguration.posRelative.direction := 0;
   // cmCathodeMainPnP2AxisZ.commandConfiguration.posAbsolute.position := 0.0;
   // cmCathodeMainPnP2AxisZ.commandConfiguration.posAbsolute.velocity := -1.0;
   // cmCathodeMainPnP2AxisZ.commandConfiguration.posAbsolute.acceleration := -1.0;
   // cmCathodeMainPnP2AxisZ.commandConfiguration.posAbsolute.deceleration := -1.0;
   // cmCathodeMainPnP2AxisZ.commandConfiguration.posAbsolute.jerk := -1.0;
   // cmCathodeMainPnP2AxisZ.commandConfiguration.posAbsolute.direction := 1;
   // cmCathodeMainPnP2AxisZ.commandConfiguration.posAbsolute.positionChangeOnTheFly := FALSE;
   // cmCathodeMainPnP2AxisZ.commandConfiguration.posAbsolute.velocityChangeOnTheFly := FALSE;
   // cmCathodeMainPnP2AxisZ.commandConfiguration.posSuperimposed.distance := 0.0;
   // cmCathodeMainPnP2AxisZ.commandConfiguration.posSuperimposed.velocityDiff := -1.0;
   // cmCathodeMainPnP2AxisZ.commandConfiguration.posSuperimposed.acceleration := -1.0;
   // cmCathodeMainPnP2AxisZ.commandConfiguration.posSuperimposed.deceleration := -1.0;
   // cmCathodeMainPnP2AxisZ.commandConfiguration.posSuperimposed.jerk := -1.0;
   // cmCathodeMainPnP2AxisZ.commandConfiguration.posSuperimposed.direction := 0;
   // cmCathodeMainPnP2AxisZ.commandConfiguration.haltSuperimposed.deceleration := -1.0;
   // cmCathodeMainPnP2AxisZ.commandConfiguration.haltSuperimposed.jerk := -1.0;
   // cmCathodeMainPnP2AxisZ.commandConfiguration.haltSuperimposed.abortAcceleration := FALSE;
   // cmCathodeMainPnP2AxisZ.commandConfiguration.gearInRelative.ratioNumerator := 1;
   // cmCathodeMainPnP2AxisZ.commandConfiguration.gearInRelative.ratioDenominator := 1;
   // cmCathodeMainPnP2AxisZ.commandConfiguration.gearInRelative.acceleration := -1.0;
   // cmCathodeMainPnP2AxisZ.commandConfiguration.gearInRelative.deceleration := -1.0;
   // cmCathodeMainPnP2AxisZ.commandConfiguration.gearInRelative.jerk := -1.0;
   // cmCathodeMainPnP2AxisZ.commandConfiguration.gearInRelative.ratioChangeOnTheFly := FALSE;
   // cmCathodeMainPnP2AxisZ.commandConfiguration.gearInAbsolute.ratioNumerator := 1;
   // cmCathodeMainPnP2AxisZ.commandConfiguration.gearInAbsolute.ratioDenominator := 1;
   // cmCathodeMainPnP2AxisZ.commandConfiguration.gearInAbsolute.masterSyncPosition := 0.0;
   // cmCathodeMainPnP2AxisZ.commandConfiguration.gearInAbsolute.slaveSyncPosition := 0.0;
   // cmCathodeMainPnP2AxisZ.commandConfiguration.gearInAbsolute.syncProfileReference := 1;
   // cmCathodeMainPnP2AxisZ.commandConfiguration.gearInAbsolute.masterStartDistance := 0.0;
   // cmCathodeMainPnP2AxisZ.commandConfiguration.gearInAbsolute.velocity := -1.0;
   // cmCathodeMainPnP2AxisZ.commandConfiguration.gearInAbsolute.acceleration := -1.0;
   // cmCathodeMainPnP2AxisZ.commandConfiguration.gearInAbsolute.deceleration := -1.0;
   // cmCathodeMainPnP2AxisZ.commandConfiguration.gearInAbsolute.jerk := -1.0;
   // cmCathodeMainPnP2AxisZ.commandConfiguration.gearInAbsolute.syncDirection := 1;
   // cmCathodeMainPnP2AxisZ.commandConfiguration.gearInAbsolute.ratioChangeOnTheFly := FALSE;
   // cmCathodeMainPnP2AxisZ.commandConfiguration.gearInVelocity.continuousUpdate := FALSE;
   // cmCathodeMainPnP2AxisZ.commandConfiguration.gearInVelocity.ratioNumerator := 1;
   // cmCathodeMainPnP2AxisZ.commandConfiguration.gearInVelocity.ratioDenominator := 1;
   // cmCathodeMainPnP2AxisZ.commandConfiguration.gearInVelocity.acceleration := -1.0;
   // cmCathodeMainPnP2AxisZ.commandConfiguration.gearInVelocity.deceleration := -1.0;
   // cmCathodeMainPnP2AxisZ.commandConfiguration.gearInVelocity.jerk := -1.0;
   // cmCathodeMainPnP2AxisZ.commandConfiguration.gearInVelocity.positionControlled := FALSE;
   // cmCathodeMainPnP2AxisZ.commandConfiguration.camIn.masterOffset := 0.0;
   // cmCathodeMainPnP2AxisZ.commandConfiguration.camIn.slaveOffset := 0.0;
   // cmCathodeMainPnP2AxisZ.commandConfiguration.camIn.masterScaling := 1.0;
   // cmCathodeMainPnP2AxisZ.commandConfiguration.camIn.slaveScaling := 1.0;
   // cmCathodeMainPnP2AxisZ.commandConfiguration.camIn.masterSyncPosition := 0.0;
   // cmCathodeMainPnP2AxisZ.commandConfiguration.camIn.syncProfileReference := 1;
   // cmCathodeMainPnP2AxisZ.commandConfiguration.camIn.masterStartDistance := 0.0;
   // cmCathodeMainPnP2AxisZ.commandConfiguration.camIn.velocity := -1.0;
   // cmCathodeMainPnP2AxisZ.commandConfiguration.camIn.acceleration := -1.0;
   // cmCathodeMainPnP2AxisZ.commandConfiguration.camIn.deceleration := -1.0;
   // cmCathodeMainPnP2AxisZ.commandConfiguration.camIn.jerk := -1.0;
   // cmCathodeMainPnP2AxisZ.commandConfiguration.camIn.applicationMode := 0;
   // cmCathodeMainPnP2AxisZ.commandConfiguration.camIn.syncDirection := 1;
   // cmCathodeMainPnP2AxisZ.commandConfiguration.gearOutCamOut.slavePosition := 0.0;
   // cmCathodeMainPnP2AxisZ.commandConfiguration.gearOutCamOut.syncProfileReference := 1;
   // cmCathodeMainPnP2AxisZ.commandConfiguration.gearOutCamOut.masterStopDistance := 0.0;
   // cmCathodeMainPnP2AxisZ.commandConfiguration.gearOutCamOut.deceleration := -1.0;
   // cmCathodeMainPnP2AxisZ.commandConfiguration.gearOutCamOut.jerk := -1.0;
   // cmCathodeMainPnP2AxisZ.commandConfiguration.gearOutCamOut.syncOutDirection := 3;
   // cmCathodeMainPnP2AxisZ.commandConfiguration.gearOutCamOut.gearOutCamOutMode := -1;
   // cmCathodeMainPnP2AxisZ.commandConfiguration.phasing.phaseShift := 0.0;
   // cmCathodeMainPnP2AxisZ.commandConfiguration.phasing.velocity := -1.0;
   // cmCathodeMainPnP2AxisZ.commandConfiguration.phasing.acceleration := -1.0;
   // cmCathodeMainPnP2AxisZ.commandConfiguration.phasing.deceleration := -1.0;
   // cmCathodeMainPnP2AxisZ.commandConfiguration.phasing.jerk := -1.0;
   // cmCathodeMainPnP2AxisZ.commandConfiguration.phasing.profileReference := 0;
   // cmCathodeMainPnP2AxisZ.commandConfiguration.phasing.phasingDistance := 0.0;
   // cmCathodeMainPnP2AxisZ.commandConfiguration.phasing.startPosition := 0.0;
   // cmCathodeMainPnP2AxisZ.commandConfiguration.phasing.direction := 3;
   // cmCathodeMainPnP2AxisZ.commandConfiguration.phasing.phaseAbsolute := TRUE;
   // cmCathodeMainPnP2AxisZ.commandConfiguration.phasing.phaseShiftChangeOnTheFly := FALSE;
   // cmCathodeMainPnP2AxisZ.commandConfiguration.offset.offset := 0.0;
   // cmCathodeMainPnP2AxisZ.commandConfiguration.offset.profileReference := 1;
   // cmCathodeMainPnP2AxisZ.commandConfiguration.offset.offsetDistance := 0.0;
   // cmCathodeMainPnP2AxisZ.commandConfiguration.offset.startPosition := 0.0;
   // cmCathodeMainPnP2AxisZ.commandConfiguration.offset.direction := 3;
   // cmCathodeMainPnP2AxisZ.commandConfiguration.offset.offsetAbsolute := TRUE;
   // cmCathodeMainPnP2AxisZ.commandConfiguration.offset.offsetChangeOnTheFly := FALSE;
   // cmCathodeMainPnP2AxisZ.commands.enableAxis := FALSE;
   // cmCathodeMainPnP2AxisZ.commands.resetAxis := FALSE;
   // cmCathodeMainPnP2AxisZ.commands.openBrake := FALSE;
   // cmCathodeMainPnP2AxisZ.commands.jogForward := FALSE;
   // cmCathodeMainPnP2AxisZ.commands.jogBackward := FALSE;
   // cmCathodeMainPnP2AxisZ.commands.moveVelocity := FALSE;
   // cmCathodeMainPnP2AxisZ.commands.stop := FALSE;
   // cmCathodeMainPnP2AxisZ.commands.fastStop := FALSE;
   // cmCathodeMainPnP2AxisZ.commands.torqueLimiting := FALSE;
   // cmCathodeMainPnP2AxisZ.commands.homing := FALSE;
   // cmCathodeMainPnP2AxisZ.commands.posRelative := FALSE;
   // cmCathodeMainPnP2AxisZ.commands.posAbsolute := FALSE;
   // cmCathodeMainPnP2AxisZ.commands.posSuperimposed := FALSE;
   // cmCathodeMainPnP2AxisZ.commands.haltSuperimposed := FALSE;
   // cmCathodeMainPnP2AxisZ.commands.selectSetPosition := -1;
   // cmCathodeMainPnP2AxisZ.commands.reset := FALSE;
   // cmCathodeMainPnP2AxisZ.monitoring.valid := FALSE;
   // cmCathodeMainPnP2AxisZ.monitoring.busy := TRUE;
   // cmCathodeMainPnP2AxisZ.monitoring.error := TRUE;
   // cmCathodeMainPnP2AxisZ.monitoring.status := 16#8600;
   // cmCathodeMainPnP2AxisZ.monitoring.subfunctionStatus := 16#8001;
   // cmCathodeMainPnP2AxisZ.monitoring.axisEnabled := FALSE;
   // cmCathodeMainPnP2AxisZ.monitoring.resetActive := FALSE;
   // cmCathodeMainPnP2AxisZ.monitoring.inVelocity := FALSE;
   // cmCathodeMainPnP2AxisZ.monitoring.inLimitation := FALSE;
   // cmCathodeMainPnP2AxisZ.monitoring.inClamping := FALSE;
   // cmCathodeMainPnP2AxisZ.monitoring.startSync := FALSE;
   // cmCathodeMainPnP2AxisZ.monitoring.inSync := FALSE;
   // cmCathodeMainPnP2AxisZ.monitoring.inSimulation := FALSE;
   // cmCathodeMainPnP2AxisZ.monitoring.jogSelected := FALSE;
   // cmCathodeMainPnP2AxisZ.monitoring.moveVelocitySelected := FALSE;
   // cmCathodeMainPnP2AxisZ.monitoring.stopSelected := FALSE;
   // cmCathodeMainPnP2AxisZ.monitoring.fastStopSelected := FALSE;
   // cmCathodeMainPnP2AxisZ.monitoring.torqueLimitingSelected := FALSE;
   // cmCathodeMainPnP2AxisZ.monitoring.homingSelected := FALSE;
   // cmCathodeMainPnP2AxisZ.monitoring.posRelativeSelected := FALSE;
   // cmCathodeMainPnP2AxisZ.monitoring.posAbsoluteSelected := FALSE;
   // cmCathodeMainPnP2AxisZ.monitoring.posSuperimposedSelected := FALSE;
   // cmCathodeMainPnP2AxisZ.monitoring.haltSuperimposedSelected := FALSE;
   // cmCathodeMainPnP2AxisZ.monitoring.commandBusy := FALSE;
   // cmCathodeMainPnP2AxisZ.monitoring.commandDone := FALSE;
   // cmCathodeMainPnP2AxisZ.monitoring.commandAborted := FALSE;
   // cmCathodeMainPnP2AxisZ.monitoring.homingCommandBusy := FALSE;
   // cmCathodeMainPnP2AxisZ.monitoring.homingCommandDone := FALSE;
   // cmCathodeMainPnP2AxisZ.monitoring.homingCommandAborted := FALSE;
   // cmCathodeMainPnP2AxisZ.monitoring.superimposedBusy := FALSE;
   // cmCathodeMainPnP2AxisZ.monitoring.superimposedDone := FALSE;
   // cmCathodeMainPnP2AxisZ.monitoring.superimposedAborted := FALSE;
   // cmCathodeMainPnP2AxisZ.monitoring.actualPosition := 2.382;
   // cmCathodeMainPnP2AxisZ.monitoring.actualSpeed := 0.0;
   // cmCathodeMainPnP2AxisZ.monitoring.speedUnit := 1062;
   // cmCathodeMainPnP2AxisZ.monitoring.positionUnit := 1013;
   // cmCathodeMainPnP2AxisZ.monitoring.axisType := 1;
   // cmCathodeMainPnP2AxisZ.monitoring.interlockGeneralOut := TRUE;
   // cmCathodeMainPnP2AxisZ.monitoring.interlockJogForwardOut := TRUE;
   // cmCathodeMainPnP2AxisZ.monitoring.interlockJogBackwardOut := TRUE;
   // cmCathodeAlignTableAxisX.commandConfiguration.generalSettings.stopOnError := TRUE;
   // cmCathodeAlignTableAxisX.commandConfiguration.generalSettings.resetWithRestart := FALSE;
   // cmCathodeAlignTableAxisX.commandConfiguration.generalSettings.abortWaitingSyncCmd := TRUE;
   // cmCathodeAlignTableAxisX.commandConfiguration.power.startMode := 1;
   // cmCathodeAlignTableAxisX.commandConfiguration.power.stopMode := 0;
   // cmCathodeAlignTableAxisX.commandConfiguration.power.syncMotionSimulation := FALSE;
   // cmCathodeAlignTableAxisX.commandConfiguration.power.syncMotionSimulationExtendedMode := -1;
   // cmCathodeAlignTableAxisX.commandConfiguration.jog.velocity := 0.0;
   // cmCathodeAlignTableAxisX.commandConfiguration.jog.acceleration := -1.0;
   // cmCathodeAlignTableAxisX.commandConfiguration.jog.deceleration := -1.0;
   // cmCathodeAlignTableAxisX.commandConfiguration.jog.jerk := -1.0;
   // cmCathodeAlignTableAxisX.commandConfiguration.jog.positionControlled := TRUE;
   // cmCathodeAlignTableAxisX.commandConfiguration.jog.increment := 0.0;
   // cmCathodeAlignTableAxisX.commandConfiguration.jog.mode := 0;
   // cmCathodeAlignTableAxisX.commandConfiguration.moveVelocity.velocity := 0.0;
   // cmCathodeAlignTableAxisX.commandConfiguration.moveVelocity.acceleration := -1.0;
   // cmCathodeAlignTableAxisX.commandConfiguration.moveVelocity.deceleration := -1.0;
   // cmCathodeAlignTableAxisX.commandConfiguration.moveVelocity.jerk := -1.0;
   // cmCathodeAlignTableAxisX.commandConfiguration.moveVelocity.direction := 0;
   // cmCathodeAlignTableAxisX.commandConfiguration.moveVelocity.positionControlled := TRUE;
   // cmCathodeAlignTableAxisX.commandConfiguration.moveVelocity.velocityChangeOnTheFly := FALSE;
   // cmCathodeAlignTableAxisX.commandConfiguration.stop.deceleration := -1.0;
   // cmCathodeAlignTableAxisX.commandConfiguration.stop.jerk := -1.0;
   // cmCathodeAlignTableAxisX.commandConfiguration.stop.abortAcceleration := FALSE;
   // cmCathodeAlignTableAxisX.commandConfiguration.fastStop.deceleration := -1.0;
   // cmCathodeAlignTableAxisX.commandConfiguration.fastStop.jerk := -1.0;
   // cmCathodeAlignTableAxisX.commandConfiguration.fastStop.abortAcceleration := FALSE;
   // cmCathodeAlignTableAxisX.commandConfiguration.fastStop.replaceStopPossible := FALSE;
   // cmCathodeAlignTableAxisX.commandConfiguration.torqueLimiting.limit := -1.0;
   // cmCathodeAlignTableAxisX.commandConfiguration.torqueLimiting.mode := 0;
   // cmCathodeAlignTableAxisX.commandConfiguration.homing.position := 0.0;
   // cmCathodeAlignTableAxisX.commandConfiguration.homing.mode := 0;
   // cmCathodeAlignTableAxisX.commandConfiguration.homing.sensor := 0;
   // cmCathodeAlignTableAxisX.commandConfiguration.homing.extendedMode := -1;
   // cmCathodeAlignTableAxisX.commandConfiguration.homing.extendedModeTorqueLimit := 0.0;
   // cmCathodeAlignTableAxisX.commandConfiguration.homing.extendedModeTargetPosition := 0.0;
   // cmCathodeAlignTableAxisX.commandConfiguration.posRelative.distance := 0.0;
   // cmCathodeAlignTableAxisX.commandConfiguration.posRelative.velocity := -1.0;
   // cmCathodeAlignTableAxisX.commandConfiguration.posRelative.acceleration := -1.0;
   // cmCathodeAlignTableAxisX.commandConfiguration.posRelative.deceleration := -1.0;
   // cmCathodeAlignTableAxisX.commandConfiguration.posRelative.jerk := -1.0;
   // cmCathodeAlignTableAxisX.commandConfiguration.posRelative.direction := 0;
   // cmCathodeAlignTableAxisX.commandConfiguration.posAbsolute.position := 0.0;
   // cmCathodeAlignTableAxisX.commandConfiguration.posAbsolute.velocity := -1.0;
   // cmCathodeAlignTableAxisX.commandConfiguration.posAbsolute.acceleration := -1.0;
   // cmCathodeAlignTableAxisX.commandConfiguration.posAbsolute.deceleration := -1.0;
   // cmCathodeAlignTableAxisX.commandConfiguration.posAbsolute.jerk := -1.0;
   // cmCathodeAlignTableAxisX.commandConfiguration.posAbsolute.direction := 1;
   // cmCathodeAlignTableAxisX.commandConfiguration.posAbsolute.positionChangeOnTheFly := FALSE;
   // cmCathodeAlignTableAxisX.commandConfiguration.posAbsolute.velocityChangeOnTheFly := FALSE;
   // cmCathodeAlignTableAxisX.commandConfiguration.posSuperimposed.distance := 0.0;
   // cmCathodeAlignTableAxisX.commandConfiguration.posSuperimposed.velocityDiff := -1.0;
   // cmCathodeAlignTableAxisX.commandConfiguration.posSuperimposed.acceleration := -1.0;
   // cmCathodeAlignTableAxisX.commandConfiguration.posSuperimposed.deceleration := -1.0;
   // cmCathodeAlignTableAxisX.commandConfiguration.posSuperimposed.jerk := -1.0;
   // cmCathodeAlignTableAxisX.commandConfiguration.posSuperimposed.direction := 0;
   // cmCathodeAlignTableAxisX.commandConfiguration.haltSuperimposed.deceleration := -1.0;
   // cmCathodeAlignTableAxisX.commandConfiguration.haltSuperimposed.jerk := -1.0;
   // cmCathodeAlignTableAxisX.commandConfiguration.haltSuperimposed.abortAcceleration := FALSE;
   // cmCathodeAlignTableAxisX.commandConfiguration.gearInRelative.ratioNumerator := 1;
   // cmCathodeAlignTableAxisX.commandConfiguration.gearInRelative.ratioDenominator := 1;
   // cmCathodeAlignTableAxisX.commandConfiguration.gearInRelative.acceleration := -1.0;
   // cmCathodeAlignTableAxisX.commandConfiguration.gearInRelative.deceleration := -1.0;
   // cmCathodeAlignTableAxisX.commandConfiguration.gearInRelative.jerk := -1.0;
   // cmCathodeAlignTableAxisX.commandConfiguration.gearInRelative.ratioChangeOnTheFly := FALSE;
   // cmCathodeAlignTableAxisX.commandConfiguration.gearInAbsolute.ratioNumerator := 1;
   // cmCathodeAlignTableAxisX.commandConfiguration.gearInAbsolute.ratioDenominator := 1;
   // cmCathodeAlignTableAxisX.commandConfiguration.gearInAbsolute.masterSyncPosition := 0.0;
   // cmCathodeAlignTableAxisX.commandConfiguration.gearInAbsolute.slaveSyncPosition := 0.0;
   // cmCathodeAlignTableAxisX.commandConfiguration.gearInAbsolute.syncProfileReference := 1;
   // cmCathodeAlignTableAxisX.commandConfiguration.gearInAbsolute.masterStartDistance := 0.0;
   // cmCathodeAlignTableAxisX.commandConfiguration.gearInAbsolute.velocity := -1.0;
   // cmCathodeAlignTableAxisX.commandConfiguration.gearInAbsolute.acceleration := -1.0;
   // cmCathodeAlignTableAxisX.commandConfiguration.gearInAbsolute.deceleration := -1.0;
   // cmCathodeAlignTableAxisX.commandConfiguration.gearInAbsolute.jerk := -1.0;
   // cmCathodeAlignTableAxisX.commandConfiguration.gearInAbsolute.syncDirection := 1;
   // cmCathodeAlignTableAxisX.commandConfiguration.gearInAbsolute.ratioChangeOnTheFly := FALSE;
   // cmCathodeAlignTableAxisX.commandConfiguration.gearInVelocity.continuousUpdate := FALSE;
   // cmCathodeAlignTableAxisX.commandConfiguration.gearInVelocity.ratioNumerator := 1;
   // cmCathodeAlignTableAxisX.commandConfiguration.gearInVelocity.ratioDenominator := 1;
   // cmCathodeAlignTableAxisX.commandConfiguration.gearInVelocity.acceleration := -1.0;
   // cmCathodeAlignTableAxisX.commandConfiguration.gearInVelocity.deceleration := -1.0;
   // cmCathodeAlignTableAxisX.commandConfiguration.gearInVelocity.jerk := -1.0;
   // cmCathodeAlignTableAxisX.commandConfiguration.gearInVelocity.positionControlled := FALSE;
   // cmCathodeAlignTableAxisX.commandConfiguration.camIn.masterOffset := 0.0;
   // cmCathodeAlignTableAxisX.commandConfiguration.camIn.slaveOffset := 0.0;
   // cmCathodeAlignTableAxisX.commandConfiguration.camIn.masterScaling := 1.0;
   // cmCathodeAlignTableAxisX.commandConfiguration.camIn.slaveScaling := 1.0;
   // cmCathodeAlignTableAxisX.commandConfiguration.camIn.masterSyncPosition := 0.0;
   // cmCathodeAlignTableAxisX.commandConfiguration.camIn.syncProfileReference := 1;
   // cmCathodeAlignTableAxisX.commandConfiguration.camIn.masterStartDistance := 0.0;
   // cmCathodeAlignTableAxisX.commandConfiguration.camIn.velocity := -1.0;
   // cmCathodeAlignTableAxisX.commandConfiguration.camIn.acceleration := -1.0;
   // cmCathodeAlignTableAxisX.commandConfiguration.camIn.deceleration := -1.0;
   // cmCathodeAlignTableAxisX.commandConfiguration.camIn.jerk := -1.0;
   // cmCathodeAlignTableAxisX.commandConfiguration.camIn.applicationMode := 0;
   // cmCathodeAlignTableAxisX.commandConfiguration.camIn.syncDirection := 1;
   // cmCathodeAlignTableAxisX.commandConfiguration.gearOutCamOut.slavePosition := 0.0;
   // cmCathodeAlignTableAxisX.commandConfiguration.gearOutCamOut.syncProfileReference := 1;
   // cmCathodeAlignTableAxisX.commandConfiguration.gearOutCamOut.masterStopDistance := 0.0;
   // cmCathodeAlignTableAxisX.commandConfiguration.gearOutCamOut.deceleration := -1.0;
   // cmCathodeAlignTableAxisX.commandConfiguration.gearOutCamOut.jerk := -1.0;
   // cmCathodeAlignTableAxisX.commandConfiguration.gearOutCamOut.syncOutDirection := 3;
   // cmCathodeAlignTableAxisX.commandConfiguration.gearOutCamOut.gearOutCamOutMode := -1;
   // cmCathodeAlignTableAxisX.commandConfiguration.phasing.phaseShift := 0.0;
   // cmCathodeAlignTableAxisX.commandConfiguration.phasing.velocity := -1.0;
   // cmCathodeAlignTableAxisX.commandConfiguration.phasing.acceleration := -1.0;
   // cmCathodeAlignTableAxisX.commandConfiguration.phasing.deceleration := -1.0;
   // cmCathodeAlignTableAxisX.commandConfiguration.phasing.jerk := -1.0;
   // cmCathodeAlignTableAxisX.commandConfiguration.phasing.profileReference := 0;
   // cmCathodeAlignTableAxisX.commandConfiguration.phasing.phasingDistance := 0.0;
   // cmCathodeAlignTableAxisX.commandConfiguration.phasing.startPosition := 0.0;
   // cmCathodeAlignTableAxisX.commandConfiguration.phasing.direction := 3;
   // cmCathodeAlignTableAxisX.commandConfiguration.phasing.phaseAbsolute := TRUE;
   // cmCathodeAlignTableAxisX.commandConfiguration.phasing.phaseShiftChangeOnTheFly := FALSE;
   // cmCathodeAlignTableAxisX.commandConfiguration.offset.offset := 0.0;
   // cmCathodeAlignTableAxisX.commandConfiguration.offset.profileReference := 1;
   // cmCathodeAlignTableAxisX.commandConfiguration.offset.offsetDistance := 0.0;
   // cmCathodeAlignTableAxisX.commandConfiguration.offset.startPosition := 0.0;
   // cmCathodeAlignTableAxisX.commandConfiguration.offset.direction := 3;
   // cmCathodeAlignTableAxisX.commandConfiguration.offset.offsetAbsolute := TRUE;
   // cmCathodeAlignTableAxisX.commandConfiguration.offset.offsetChangeOnTheFly := FALSE;
   // cmCathodeAlignTableAxisX.commands.enableAxis := FALSE;
   // cmCathodeAlignTableAxisX.commands.resetAxis := FALSE;
   // cmCathodeAlignTableAxisX.commands.openBrake := FALSE;
   // cmCathodeAlignTableAxisX.commands.jogForward := FALSE;
   // cmCathodeAlignTableAxisX.commands.jogBackward := FALSE;
   // cmCathodeAlignTableAxisX.commands.moveVelocity := FALSE;
   // cmCathodeAlignTableAxisX.commands.stop := FALSE;
   // cmCathodeAlignTableAxisX.commands.fastStop := FALSE;
   // cmCathodeAlignTableAxisX.commands.torqueLimiting := FALSE;
   // cmCathodeAlignTableAxisX.commands.homing := FALSE;
   // cmCathodeAlignTableAxisX.commands.posRelative := FALSE;
   // cmCathodeAlignTableAxisX.commands.posAbsolute := FALSE;
   // cmCathodeAlignTableAxisX.commands.posSuperimposed := FALSE;
   // cmCathodeAlignTableAxisX.commands.haltSuperimposed := FALSE;
   // cmCathodeAlignTableAxisX.commands.selectSetPosition := -1;
   // cmCathodeAlignTableAxisX.commands.reset := FALSE;
   // cmCathodeAlignTableAxisX.monitoring.valid := FALSE;
   // cmCathodeAlignTableAxisX.monitoring.busy := TRUE;
   // cmCathodeAlignTableAxisX.monitoring.error := TRUE;
   // cmCathodeAlignTableAxisX.monitoring.status := 16#8600;
   // cmCathodeAlignTableAxisX.monitoring.subfunctionStatus := 16#8001;
   // cmCathodeAlignTableAxisX.monitoring.axisEnabled := FALSE;
   // cmCathodeAlignTableAxisX.monitoring.resetActive := FALSE;
   // cmCathodeAlignTableAxisX.monitoring.inVelocity := FALSE;
   // cmCathodeAlignTableAxisX.monitoring.inLimitation := FALSE;
   // cmCathodeAlignTableAxisX.monitoring.inClamping := FALSE;
   // cmCathodeAlignTableAxisX.monitoring.startSync := FALSE;
   // cmCathodeAlignTableAxisX.monitoring.inSync := FALSE;
   // cmCathodeAlignTableAxisX.monitoring.inSimulation := FALSE;
   // cmCathodeAlignTableAxisX.monitoring.jogSelected := FALSE;
   // cmCathodeAlignTableAxisX.monitoring.moveVelocitySelected := FALSE;
   // cmCathodeAlignTableAxisX.monitoring.stopSelected := FALSE;
   // cmCathodeAlignTableAxisX.monitoring.fastStopSelected := FALSE;
   // cmCathodeAlignTableAxisX.monitoring.torqueLimitingSelected := FALSE;
   // cmCathodeAlignTableAxisX.monitoring.homingSelected := FALSE;
   // cmCathodeAlignTableAxisX.monitoring.posRelativeSelected := FALSE;
   // cmCathodeAlignTableAxisX.monitoring.posAbsoluteSelected := FALSE;
   // cmCathodeAlignTableAxisX.monitoring.posSuperimposedSelected := FALSE;
   // cmCathodeAlignTableAxisX.monitoring.haltSuperimposedSelected := FALSE;
   // cmCathodeAlignTableAxisX.monitoring.commandBusy := FALSE;
   // cmCathodeAlignTableAxisX.monitoring.commandDone := FALSE;
   // cmCathodeAlignTableAxisX.monitoring.commandAborted := FALSE;
   // cmCathodeAlignTableAxisX.monitoring.homingCommandBusy := FALSE;
   // cmCathodeAlignTableAxisX.monitoring.homingCommandDone := FALSE;
   // cmCathodeAlignTableAxisX.monitoring.homingCommandAborted := FALSE;
   // cmCathodeAlignTableAxisX.monitoring.superimposedBusy := FALSE;
   // cmCathodeAlignTableAxisX.monitoring.superimposedDone := FALSE;
   // cmCathodeAlignTableAxisX.monitoring.superimposedAborted := FALSE;
   // cmCathodeAlignTableAxisX.monitoring.actualPosition := -0.929;
   // cmCathodeAlignTableAxisX.monitoring.actualSpeed := 0.0;
   // cmCathodeAlignTableAxisX.monitoring.speedUnit := 1062;
   // cmCathodeAlignTableAxisX.monitoring.positionUnit := 1013;
   // cmCathodeAlignTableAxisX.monitoring.axisType := 1;
   // cmCathodeAlignTableAxisX.monitoring.interlockGeneralOut := TRUE;
   // cmCathodeAlignTableAxisX.monitoring.interlockJogForwardOut := TRUE;
   // cmCathodeAlignTableAxisX.monitoring.interlockJogBackwardOut := TRUE;
   // cmCathodeAlignTableAxisY1.commandConfiguration.generalSettings.stopOnError := TRUE;
   // cmCathodeAlignTableAxisY1.commandConfiguration.generalSettings.resetWithRestart := FALSE;
   // cmCathodeAlignTableAxisY1.commandConfiguration.generalSettings.abortWaitingSyncCmd := TRUE;
   // cmCathodeAlignTableAxisY1.commandConfiguration.power.startMode := 1;
   // cmCathodeAlignTableAxisY1.commandConfiguration.power.stopMode := 0;
   // cmCathodeAlignTableAxisY1.commandConfiguration.power.syncMotionSimulation := FALSE;
   // cmCathodeAlignTableAxisY1.commandConfiguration.power.syncMotionSimulationExtendedMode := -1;
   // cmCathodeAlignTableAxisY1.commandConfiguration.jog.velocity := 0.0;
   // cmCathodeAlignTableAxisY1.commandConfiguration.jog.acceleration := -1.0;
   // cmCathodeAlignTableAxisY1.commandConfiguration.jog.deceleration := -1.0;
   // cmCathodeAlignTableAxisY1.commandConfiguration.jog.jerk := -1.0;
   // cmCathodeAlignTableAxisY1.commandConfiguration.jog.positionControlled := TRUE;
   // cmCathodeAlignTableAxisY1.commandConfiguration.jog.increment := 0.0;
   // cmCathodeAlignTableAxisY1.commandConfiguration.jog.mode := 0;
   // cmCathodeAlignTableAxisY1.commandConfiguration.moveVelocity.velocity := 0.0;
   // cmCathodeAlignTableAxisY1.commandConfiguration.moveVelocity.acceleration := -1.0;
   // cmCathodeAlignTableAxisY1.commandConfiguration.moveVelocity.deceleration := -1.0;
   // cmCathodeAlignTableAxisY1.commandConfiguration.moveVelocity.jerk := -1.0;
   // cmCathodeAlignTableAxisY1.commandConfiguration.moveVelocity.direction := 0;
   // cmCathodeAlignTableAxisY1.commandConfiguration.moveVelocity.positionControlled := TRUE;
   // cmCathodeAlignTableAxisY1.commandConfiguration.moveVelocity.velocityChangeOnTheFly := FALSE;
   // cmCathodeAlignTableAxisY1.commandConfiguration.stop.deceleration := -1.0;
   // cmCathodeAlignTableAxisY1.commandConfiguration.stop.jerk := -1.0;
   // cmCathodeAlignTableAxisY1.commandConfiguration.stop.abortAcceleration := FALSE;
   // cmCathodeAlignTableAxisY1.commandConfiguration.fastStop.deceleration := -1.0;
   // cmCathodeAlignTableAxisY1.commandConfiguration.fastStop.jerk := -1.0;
   // cmCathodeAlignTableAxisY1.commandConfiguration.fastStop.abortAcceleration := FALSE;
   // cmCathodeAlignTableAxisY1.commandConfiguration.fastStop.replaceStopPossible := FALSE;
   // cmCathodeAlignTableAxisY1.commandConfiguration.torqueLimiting.limit := -1.0;
   // cmCathodeAlignTableAxisY1.commandConfiguration.torqueLimiting.mode := 0;
   // cmCathodeAlignTableAxisY1.commandConfiguration.homing.position := 0.0;
   // cmCathodeAlignTableAxisY1.commandConfiguration.homing.mode := 0;
   // cmCathodeAlignTableAxisY1.commandConfiguration.homing.sensor := 0;
   // cmCathodeAlignTableAxisY1.commandConfiguration.homing.extendedMode := -1;
   // cmCathodeAlignTableAxisY1.commandConfiguration.homing.extendedModeTorqueLimit := 0.0;
   // cmCathodeAlignTableAxisY1.commandConfiguration.homing.extendedModeTargetPosition := 0.0;
   // cmCathodeAlignTableAxisY1.commandConfiguration.posRelative.distance := 0.0;
   // cmCathodeAlignTableAxisY1.commandConfiguration.posRelative.velocity := -1.0;
   // cmCathodeAlignTableAxisY1.commandConfiguration.posRelative.acceleration := -1.0;
   // cmCathodeAlignTableAxisY1.commandConfiguration.posRelative.deceleration := -1.0;
   // cmCathodeAlignTableAxisY1.commandConfiguration.posRelative.jerk := -1.0;
   // cmCathodeAlignTableAxisY1.commandConfiguration.posRelative.direction := 0;
   // cmCathodeAlignTableAxisY1.commandConfiguration.posAbsolute.position := 0.0;
   // cmCathodeAlignTableAxisY1.commandConfiguration.posAbsolute.velocity := -1.0;
   // cmCathodeAlignTableAxisY1.commandConfiguration.posAbsolute.acceleration := -1.0;
   // cmCathodeAlignTableAxisY1.commandConfiguration.posAbsolute.deceleration := -1.0;
   // cmCathodeAlignTableAxisY1.commandConfiguration.posAbsolute.jerk := -1.0;
   // cmCathodeAlignTableAxisY1.commandConfiguration.posAbsolute.direction := 1;
   // cmCathodeAlignTableAxisY1.commandConfiguration.posAbsolute.positionChangeOnTheFly := FALSE;
   // cmCathodeAlignTableAxisY1.commandConfiguration.posAbsolute.velocityChangeOnTheFly := FALSE;
   // cmCathodeAlignTableAxisY1.commandConfiguration.posSuperimposed.distance := 0.0;
   // cmCathodeAlignTableAxisY1.commandConfiguration.posSuperimposed.velocityDiff := -1.0;
   // cmCathodeAlignTableAxisY1.commandConfiguration.posSuperimposed.acceleration := -1.0;
   // cmCathodeAlignTableAxisY1.commandConfiguration.posSuperimposed.deceleration := -1.0;
   // cmCathodeAlignTableAxisY1.commandConfiguration.posSuperimposed.jerk := -1.0;
   // cmCathodeAlignTableAxisY1.commandConfiguration.posSuperimposed.direction := 0;
   // cmCathodeAlignTableAxisY1.commandConfiguration.haltSuperimposed.deceleration := -1.0;
   // cmCathodeAlignTableAxisY1.commandConfiguration.haltSuperimposed.jerk := -1.0;
   // cmCathodeAlignTableAxisY1.commandConfiguration.haltSuperimposed.abortAcceleration := FALSE;
   // cmCathodeAlignTableAxisY1.commandConfiguration.gearInRelative.ratioNumerator := 1;
   // cmCathodeAlignTableAxisY1.commandConfiguration.gearInRelative.ratioDenominator := 1;
   // cmCathodeAlignTableAxisY1.commandConfiguration.gearInRelative.acceleration := -1.0;
   // cmCathodeAlignTableAxisY1.commandConfiguration.gearInRelative.deceleration := -1.0;
   // cmCathodeAlignTableAxisY1.commandConfiguration.gearInRelative.jerk := -1.0;
   // cmCathodeAlignTableAxisY1.commandConfiguration.gearInRelative.ratioChangeOnTheFly := FALSE;
   // cmCathodeAlignTableAxisY1.commandConfiguration.gearInAbsolute.ratioNumerator := 1;
   // cmCathodeAlignTableAxisY1.commandConfiguration.gearInAbsolute.ratioDenominator := 1;
   // cmCathodeAlignTableAxisY1.commandConfiguration.gearInAbsolute.masterSyncPosition := 0.0;
   // cmCathodeAlignTableAxisY1.commandConfiguration.gearInAbsolute.slaveSyncPosition := 0.0;
   // cmCathodeAlignTableAxisY1.commandConfiguration.gearInAbsolute.syncProfileReference := 1;
   // cmCathodeAlignTableAxisY1.commandConfiguration.gearInAbsolute.masterStartDistance := 0.0;
   // cmCathodeAlignTableAxisY1.commandConfiguration.gearInAbsolute.velocity := -1.0;
   // cmCathodeAlignTableAxisY1.commandConfiguration.gearInAbsolute.acceleration := -1.0;
   // cmCathodeAlignTableAxisY1.commandConfiguration.gearInAbsolute.deceleration := -1.0;
   // cmCathodeAlignTableAxisY1.commandConfiguration.gearInAbsolute.jerk := -1.0;
   // cmCathodeAlignTableAxisY1.commandConfiguration.gearInAbsolute.syncDirection := 1;
   // cmCathodeAlignTableAxisY1.commandConfiguration.gearInAbsolute.ratioChangeOnTheFly := FALSE;
   // cmCathodeAlignTableAxisY1.commandConfiguration.gearInVelocity.continuousUpdate := FALSE;
   // cmCathodeAlignTableAxisY1.commandConfiguration.gearInVelocity.ratioNumerator := 1;
   // cmCathodeAlignTableAxisY1.commandConfiguration.gearInVelocity.ratioDenominator := 1;
   // cmCathodeAlignTableAxisY1.commandConfiguration.gearInVelocity.acceleration := -1.0;
   // cmCathodeAlignTableAxisY1.commandConfiguration.gearInVelocity.deceleration := -1.0;
   // cmCathodeAlignTableAxisY1.commandConfiguration.gearInVelocity.jerk := -1.0;
   // cmCathodeAlignTableAxisY1.commandConfiguration.gearInVelocity.positionControlled := FALSE;
   // cmCathodeAlignTableAxisY1.commandConfiguration.camIn.masterOffset := 0.0;
   // cmCathodeAlignTableAxisY1.commandConfiguration.camIn.slaveOffset := 0.0;
   // cmCathodeAlignTableAxisY1.commandConfiguration.camIn.masterScaling := 1.0;
   // cmCathodeAlignTableAxisY1.commandConfiguration.camIn.slaveScaling := 1.0;
   // cmCathodeAlignTableAxisY1.commandConfiguration.camIn.masterSyncPosition := 0.0;
   // cmCathodeAlignTableAxisY1.commandConfiguration.camIn.syncProfileReference := 1;
   // cmCathodeAlignTableAxisY1.commandConfiguration.camIn.masterStartDistance := 0.0;
   // cmCathodeAlignTableAxisY1.commandConfiguration.camIn.velocity := -1.0;
   // cmCathodeAlignTableAxisY1.commandConfiguration.camIn.acceleration := -1.0;
   // cmCathodeAlignTableAxisY1.commandConfiguration.camIn.deceleration := -1.0;
   // cmCathodeAlignTableAxisY1.commandConfiguration.camIn.jerk := -1.0;
   // cmCathodeAlignTableAxisY1.commandConfiguration.camIn.applicationMode := 0;
   // cmCathodeAlignTableAxisY1.commandConfiguration.camIn.syncDirection := 1;
   // cmCathodeAlignTableAxisY1.commandConfiguration.gearOutCamOut.slavePosition := 0.0;
   // cmCathodeAlignTableAxisY1.commandConfiguration.gearOutCamOut.syncProfileReference := 1;
   // cmCathodeAlignTableAxisY1.commandConfiguration.gearOutCamOut.masterStopDistance := 0.0;
   // cmCathodeAlignTableAxisY1.commandConfiguration.gearOutCamOut.deceleration := -1.0;
   // cmCathodeAlignTableAxisY1.commandConfiguration.gearOutCamOut.jerk := -1.0;
   // cmCathodeAlignTableAxisY1.commandConfiguration.gearOutCamOut.syncOutDirection := 3;
   // cmCathodeAlignTableAxisY1.commandConfiguration.gearOutCamOut.gearOutCamOutMode := -1;
   // cmCathodeAlignTableAxisY1.commandConfiguration.phasing.phaseShift := 0.0;
   // cmCathodeAlignTableAxisY1.commandConfiguration.phasing.velocity := -1.0;
   // cmCathodeAlignTableAxisY1.commandConfiguration.phasing.acceleration := -1.0;
   // cmCathodeAlignTableAxisY1.commandConfiguration.phasing.deceleration := -1.0;
   // cmCathodeAlignTableAxisY1.commandConfiguration.phasing.jerk := -1.0;
   // cmCathodeAlignTableAxisY1.commandConfiguration.phasing.profileReference := 0;
   // cmCathodeAlignTableAxisY1.commandConfiguration.phasing.phasingDistance := 0.0;
   // cmCathodeAlignTableAxisY1.commandConfiguration.phasing.startPosition := 0.0;
   // cmCathodeAlignTableAxisY1.commandConfiguration.phasing.direction := 3;
   // cmCathodeAlignTableAxisY1.commandConfiguration.phasing.phaseAbsolute := TRUE;
   // cmCathodeAlignTableAxisY1.commandConfiguration.phasing.phaseShiftChangeOnTheFly := FALSE;
   // cmCathodeAlignTableAxisY1.commandConfiguration.offset.offset := 0.0;
   // cmCathodeAlignTableAxisY1.commandConfiguration.offset.profileReference := 1;
